(* Visualisation graf
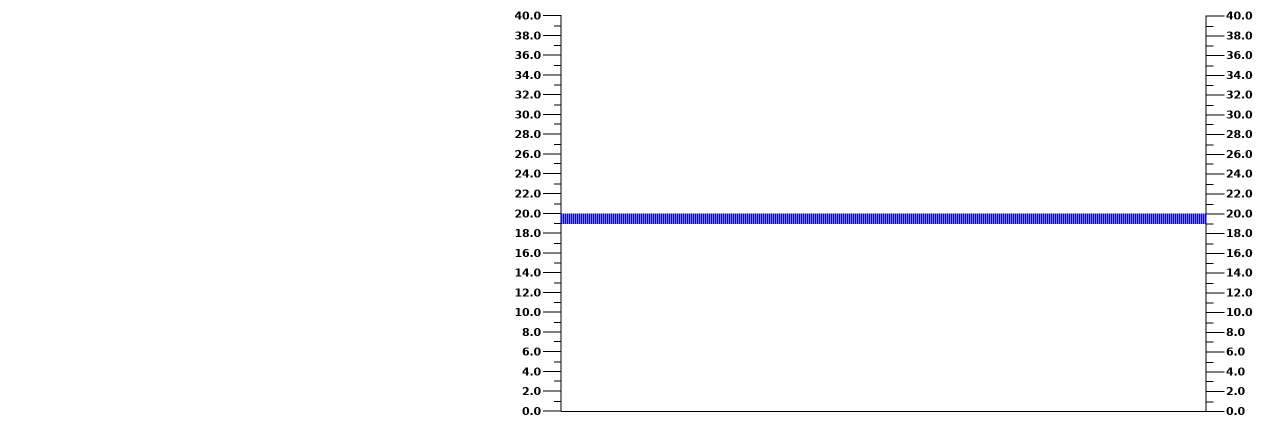
group at (130,90)-(861,501)
  rectangle at (0,8)-(1,9): text "{ExtendedElement},Visu\ElementDLL.ete,2,@Histogramm,731,411,PLC_PRG.test,,%.1f,1,2,0,40,0,0,0,0,0,0,0,-13,16,700,Arial,0,0,255,255,0,0,0,0,0,1,0.9,0_360,0,1,0,"
  rectangle at (0,411)-(25,427): text "0.0"
  rectangle at (706,411)-(731,427): text "0.0"
  rectangle at (0,390)-(25,406): text "2.0"
  rectangle at (706,390)-(731,406): text "2.0"
  rectangle at (0,370)-(25,386): text "4.0"
  rectangle at (706,370)-(731,386): text "4.0"
  rectangle at (0,349)-(25,365): text "6.0"
  rectangle at (706,349)-(731,365): text "6.0"
  rectangle at (0,329)-(25,345): text "8.0"
  rectangle at (706,329)-(731,345): text "8.0"
  rectangle at (0,308)-(25,324): text "10.0"
  rectangle at (706,308)-(731,324): text "10.0"
  rectangle at (0,288)-(25,304): text "12.0"
  rectangle at (706,288)-(731,304): text "12.0"
  rectangle at (0,267)-(25,283): text "14.0"
  rectangle at (706,267)-(731,283): text "14.0"
  rectangle at (0,247)-(25,263): text "16.0"
  rectangle at (706,247)-(731,263): text "16.0"
  rectangle at (0,226)-(25,242): text "18.0"
  rectangle at (706,226)-(731,242): text "18.0"
  rectangle at (0,206)-(25,222): text "20.0"
  rectangle at (706,206)-(731,222): text "20.0"
  rectangle at (0,185)-(25,201): text "22.0"
  rectangle at (706,185)-(731,201): text "22.0"
  rectangle at (0,164)-(25,180): text "24.0"
  rectangle at (706,164)-(731,180): text "24.0"
  rectangle at (0,144)-(25,160): text "26.0"
  rectangle at (706,144)-(731,160): text "26.0"
  rectangle at (0,123)-(25,139): text "28.0"
  rectangle at (706,123)-(731,139): text "28.0"
  rectangle at (0,103)-(25,119): text "30.0"
  rectangle at (706,103)-(731,119): text "30.0"
  rectangle at (0,82)-(25,98): text "32.0"
  rectangle at (706,82)-(731,98): text "32.0"
  rectangle at (0,62)-(25,78): text "34.0"
  rectangle at (706,62)-(731,78): text "34.0"
  rectangle at (0,41)-(25,57): text "36.0"
  rectangle at (706,41)-(731,57): text "36.0"
  rectangle at (0,21)-(25,37): text "38.0"
  rectangle at (706,21)-(731,37): text "38.0"
  rectangle at (0,0)-(25,16): text "40.0"
  rectangle at (706,0)-(731,16): text "40.0"
  rectangle at (43,214)-(44,224): alarm colour if PLC_PRG.test[0] < 0; top (-1.0 *  PLC_PRG.test[0]  +  20  ) * 10.275 + SEL( PLC_PRG.test[0] > 20 , 0.5, -0.5); bottom (-1.0 *  PLC_PRG.test[0]  +  20  ) * 10.275 + SEL( PLC_PRG.test[0] > 20 , 0.5, -0.5)
  rectangle at (45,214)-(46,224): alarm colour if PLC_PRG.test[1] < 0; top (-1.0 *  PLC_PRG.test[1]  +  20  ) * 10.275 + SEL( PLC_PRG.test[1] > 20 , 0.5, -0.5); bottom (-1.0 *  PLC_PRG.test[1]  +  20  ) * 10.275 + SEL( PLC_PRG.test[1] > 20 , 0.5, -0.5)
  rectangle at (47,214)-(48,224): alarm colour if PLC_PRG.test[2] < 0; top (-1.0 *  PLC_PRG.test[2]  +  20  ) * 10.275 + SEL( PLC_PRG.test[2] > 20 , 0.5, -0.5); bottom (-1.0 *  PLC_PRG.test[2]  +  20  ) * 10.275 + SEL( PLC_PRG.test[2] > 20 , 0.5, -0.5)
  rectangle at (49,214)-(50,224): alarm colour if PLC_PRG.test[3] < 0; top (-1.0 *  PLC_PRG.test[3]  +  20  ) * 10.275 + SEL( PLC_PRG.test[3] > 20 , 0.5, -0.5); bottom (-1.0 *  PLC_PRG.test[3]  +  20  ) * 10.275 + SEL( PLC_PRG.test[3] > 20 , 0.5, -0.5)
  rectangle at (51,214)-(52,224): alarm colour if PLC_PRG.test[4] < 0; top (-1.0 *  PLC_PRG.test[4]  +  20  ) * 10.275 + SEL( PLC_PRG.test[4] > 20 , 0.5, -0.5); bottom (-1.0 *  PLC_PRG.test[4]  +  20  ) * 10.275 + SEL( PLC_PRG.test[4] > 20 , 0.5, -0.5)
  rectangle at (53,214)-(54,224): alarm colour if PLC_PRG.test[5] < 0; top (-1.0 *  PLC_PRG.test[5]  +  20  ) * 10.275 + SEL( PLC_PRG.test[5] > 20 , 0.5, -0.5); bottom (-1.0 *  PLC_PRG.test[5]  +  20  ) * 10.275 + SEL( PLC_PRG.test[5] > 20 , 0.5, -0.5)
  rectangle at (55,214)-(56,224): alarm colour if PLC_PRG.test[6] < 0; top (-1.0 *  PLC_PRG.test[6]  +  20  ) * 10.275 + SEL( PLC_PRG.test[6] > 20 , 0.5, -0.5); bottom (-1.0 *  PLC_PRG.test[6]  +  20  ) * 10.275 + SEL( PLC_PRG.test[6] > 20 , 0.5, -0.5)
  rectangle at (57,214)-(58,224): alarm colour if PLC_PRG.test[7] < 0; top (-1.0 *  PLC_PRG.test[7]  +  20  ) * 10.275 + SEL( PLC_PRG.test[7] > 20 , 0.5, -0.5); bottom (-1.0 *  PLC_PRG.test[7]  +  20  ) * 10.275 + SEL( PLC_PRG.test[7] > 20 , 0.5, -0.5)
  rectangle at (59,214)-(60,224): alarm colour if PLC_PRG.test[8] < 0; top (-1.0 *  PLC_PRG.test[8]  +  20  ) * 10.275 + SEL( PLC_PRG.test[8] > 20 , 0.5, -0.5); bottom (-1.0 *  PLC_PRG.test[8]  +  20  ) * 10.275 + SEL( PLC_PRG.test[8] > 20 , 0.5, -0.5)
  rectangle at (61,214)-(62,224): alarm colour if PLC_PRG.test[9] < 0; top (-1.0 *  PLC_PRG.test[9]  +  20  ) * 10.275 + SEL( PLC_PRG.test[9] > 20 , 0.5, -0.5); bottom (-1.0 *  PLC_PRG.test[9]  +  20  ) * 10.275 + SEL( PLC_PRG.test[9] > 20 , 0.5, -0.5)
  rectangle at (63,214)-(64,224): alarm colour if PLC_PRG.test[10] < 0; top (-1.0 *  PLC_PRG.test[10]  +  20  ) * 10.275 + SEL( PLC_PRG.test[10] > 20 , 0.5, -0.5); bottom (-1.0 *  PLC_PRG.test[10]  +  20  ) * 10.275 + SEL( PLC_PRG.test[10] > 20 , 0.5, -0.5)
  rectangle at (65,214)-(66,224): alarm colour if PLC_PRG.test[11] < 0; top (-1.0 *  PLC_PRG.test[11]  +  20  ) * 10.275 + SEL( PLC_PRG.test[11] > 20 , 0.5, -0.5); bottom (-1.0 *  PLC_PRG.test[11]  +  20  ) * 10.275 + SEL( PLC_PRG.test[11] > 20 , 0.5, -0.5)
  rectangle at (67,214)-(68,224): alarm colour if PLC_PRG.test[12] < 0; top (-1.0 *  PLC_PRG.test[12]  +  20  ) * 10.275 + SEL( PLC_PRG.test[12] > 20 , 0.5, -0.5); bottom (-1.0 *  PLC_PRG.test[12]  +  20  ) * 10.275 + SEL( PLC_PRG.test[12] > 20 , 0.5, -0.5)
  rectangle at (69,214)-(70,224): alarm colour if PLC_PRG.test[13] < 0; top (-1.0 *  PLC_PRG.test[13]  +  20  ) * 10.275 + SEL( PLC_PRG.test[13] > 20 , 0.5, -0.5); bottom (-1.0 *  PLC_PRG.test[13]  +  20  ) * 10.275 + SEL( PLC_PRG.test[13] > 20 , 0.5, -0.5)
  rectangle at (71,214)-(72,224): alarm colour if PLC_PRG.test[14] < 0; top (-1.0 *  PLC_PRG.test[14]  +  20  ) * 10.275 + SEL( PLC_PRG.test[14] > 20 , 0.5, -0.5); bottom (-1.0 *  PLC_PRG.test[14]  +  20  ) * 10.275 + SEL( PLC_PRG.test[14] > 20 , 0.5, -0.5)
  rectangle at (73,214)-(74,224): alarm colour if PLC_PRG.test[15] < 0; top (-1.0 *  PLC_PRG.test[15]  +  20  ) * 10.275 + SEL( PLC_PRG.test[15] > 20 , 0.5, -0.5); bottom (-1.0 *  PLC_PRG.test[15]  +  20  ) * 10.275 + SEL( PLC_PRG.test[15] > 20 , 0.5, -0.5)
  rectangle at (75,214)-(76,224): alarm colour if PLC_PRG.test[16] < 0; top (-1.0 *  PLC_PRG.test[16]  +  20  ) * 10.275 + SEL( PLC_PRG.test[16] > 20 , 0.5, -0.5); bottom (-1.0 *  PLC_PRG.test[16]  +  20  ) * 10.275 + SEL( PLC_PRG.test[16] > 20 , 0.5, -0.5)
  rectangle at (77,214)-(78,224): alarm colour if PLC_PRG.test[17] < 0; top (-1.0 *  PLC_PRG.test[17]  +  20  ) * 10.275 + SEL( PLC_PRG.test[17] > 20 , 0.5, -0.5); bottom (-1.0 *  PLC_PRG.test[17]  +  20  ) * 10.275 + SEL( PLC_PRG.test[17] > 20 , 0.5, -0.5)
  rectangle at (79,214)-(80,224): alarm colour if PLC_PRG.test[18] < 0; top (-1.0 *  PLC_PRG.test[18]  +  20  ) * 10.275 + SEL( PLC_PRG.test[18] > 20 , 0.5, -0.5); bottom (-1.0 *  PLC_PRG.test[18]  +  20  ) * 10.275 + SEL( PLC_PRG.test[18] > 20 , 0.5, -0.5)
  rectangle at (81,214)-(82,224): alarm colour if PLC_PRG.test[19] < 0; top (-1.0 *  PLC_PRG.test[19]  +  20  ) * 10.275 + SEL( PLC_PRG.test[19] > 20 , 0.5, -0.5); bottom (-1.0 *  PLC_PRG.test[19]  +  20  ) * 10.275 + SEL( PLC_PRG.test[19] > 20 , 0.5, -0.5)
  rectangle at (83,214)-(84,224): alarm colour if PLC_PRG.test[20] < 0; top (-1.0 *  PLC_PRG.test[20]  +  20  ) * 10.275 + SEL( PLC_PRG.test[20] > 20 , 0.5, -0.5); bottom (-1.0 *  PLC_PRG.test[20]  +  20  ) * 10.275 + SEL( PLC_PRG.test[20] > 20 , 0.5, -0.5)
  rectangle at (85,214)-(86,224): alarm colour if PLC_PRG.test[21] < 0; top (-1.0 *  PLC_PRG.test[21]  +  20  ) * 10.275 + SEL( PLC_PRG.test[21] > 20 , 0.5, -0.5); bottom (-1.0 *  PLC_PRG.test[21]  +  20  ) * 10.275 + SEL( PLC_PRG.test[21] > 20 , 0.5, -0.5)
  rectangle at (87,214)-(88,224): alarm colour if PLC_PRG.test[22] < 0; top (-1.0 *  PLC_PRG.test[22]  +  20  ) * 10.275 + SEL( PLC_PRG.test[22] > 20 , 0.5, -0.5); bottom (-1.0 *  PLC_PRG.test[22]  +  20  ) * 10.275 + SEL( PLC_PRG.test[22] > 20 , 0.5, -0.5)
  rectangle at (89,214)-(90,224): alarm colour if PLC_PRG.test[23] < 0; top (-1.0 *  PLC_PRG.test[23]  +  20  ) * 10.275 + SEL( PLC_PRG.test[23] > 20 , 0.5, -0.5); bottom (-1.0 *  PLC_PRG.test[23]  +  20  ) * 10.275 + SEL( PLC_PRG.test[23] > 20 , 0.5, -0.5)
  rectangle at (91,214)-(92,224): alarm colour if PLC_PRG.test[24] < 0; top (-1.0 *  PLC_PRG.test[24]  +  20  ) * 10.275 + SEL( PLC_PRG.test[24] > 20 , 0.5, -0.5); bottom (-1.0 *  PLC_PRG.test[24]  +  20  ) * 10.275 + SEL( PLC_PRG.test[24] > 20 , 0.5, -0.5)
  rectangle at (93,214)-(94,224): alarm colour if PLC_PRG.test[25] < 0; top (-1.0 *  PLC_PRG.test[25]  +  20  ) * 10.275 + SEL( PLC_PRG.test[25] > 20 , 0.5, -0.5); bottom (-1.0 *  PLC_PRG.test[25]  +  20  ) * 10.275 + SEL( PLC_PRG.test[25] > 20 , 0.5, -0.5)
  rectangle at (95,214)-(96,224): alarm colour if PLC_PRG.test[26] < 0; top (-1.0 *  PLC_PRG.test[26]  +  20  ) * 10.275 + SEL( PLC_PRG.test[26] > 20 , 0.5, -0.5); bottom (-1.0 *  PLC_PRG.test[26]  +  20  ) * 10.275 + SEL( PLC_PRG.test[26] > 20 , 0.5, -0.5)
  rectangle at (97,214)-(98,224): alarm colour if PLC_PRG.test[27] < 0; top (-1.0 *  PLC_PRG.test[27]  +  20  ) * 10.275 + SEL( PLC_PRG.test[27] > 20 , 0.5, -0.5); bottom (-1.0 *  PLC_PRG.test[27]  +  20  ) * 10.275 + SEL( PLC_PRG.test[27] > 20 , 0.5, -0.5)
  rectangle at (99,214)-(100,224): alarm colour if PLC_PRG.test[28] < 0; top (-1.0 *  PLC_PRG.test[28]  +  20  ) * 10.275 + SEL( PLC_PRG.test[28] > 20 , 0.5, -0.5); bottom (-1.0 *  PLC_PRG.test[28]  +  20  ) * 10.275 + SEL( PLC_PRG.test[28] > 20 , 0.5, -0.5)
  rectangle at (101,214)-(102,224): alarm colour if PLC_PRG.test[29] < 0; top (-1.0 *  PLC_PRG.test[29]  +  20  ) * 10.275 + SEL( PLC_PRG.test[29] > 20 , 0.5, -0.5); bottom (-1.0 *  PLC_PRG.test[29]  +  20  ) * 10.275 + SEL( PLC_PRG.test[29] > 20 , 0.5, -0.5)
  rectangle at (103,214)-(104,224): alarm colour if PLC_PRG.test[30] < 0; top (-1.0 *  PLC_PRG.test[30]  +  20  ) * 10.275 + SEL( PLC_PRG.test[30] > 20 , 0.5, -0.5); bottom (-1.0 *  PLC_PRG.test[30]  +  20  ) * 10.275 + SEL( PLC_PRG.test[30] > 20 , 0.5, -0.5)
  rectangle at (105,214)-(106,224): alarm colour if PLC_PRG.test[31] < 0; top (-1.0 *  PLC_PRG.test[31]  +  20  ) * 10.275 + SEL( PLC_PRG.test[31] > 20 , 0.5, -0.5); bottom (-1.0 *  PLC_PRG.test[31]  +  20  ) * 10.275 + SEL( PLC_PRG.test[31] > 20 , 0.5, -0.5)
  rectangle at (107,214)-(108,224): alarm colour if PLC_PRG.test[32] < 0; top (-1.0 *  PLC_PRG.test[32]  +  20  ) * 10.275 + SEL( PLC_PRG.test[32] > 20 , 0.5, -0.5); bottom (-1.0 *  PLC_PRG.test[32]  +  20  ) * 10.275 + SEL( PLC_PRG.test[32] > 20 , 0.5, -0.5)
  rectangle at (109,214)-(110,224): alarm colour if PLC_PRG.test[33] < 0; top (-1.0 *  PLC_PRG.test[33]  +  20  ) * 10.275 + SEL( PLC_PRG.test[33] > 20 , 0.5, -0.5); bottom (-1.0 *  PLC_PRG.test[33]  +  20  ) * 10.275 + SEL( PLC_PRG.test[33] > 20 , 0.5, -0.5)
  rectangle at (111,214)-(112,224): alarm colour if PLC_PRG.test[34] < 0; top (-1.0 *  PLC_PRG.test[34]  +  20  ) * 10.275 + SEL( PLC_PRG.test[34] > 20 , 0.5, -0.5); bottom (-1.0 *  PLC_PRG.test[34]  +  20  ) * 10.275 + SEL( PLC_PRG.test[34] > 20 , 0.5, -0.5)
  rectangle at (113,214)-(114,224): alarm colour if PLC_PRG.test[35] < 0; top (-1.0 *  PLC_PRG.test[35]  +  20  ) * 10.275 + SEL( PLC_PRG.test[35] > 20 , 0.5, -0.5); bottom (-1.0 *  PLC_PRG.test[35]  +  20  ) * 10.275 + SEL( PLC_PRG.test[35] > 20 , 0.5, -0.5)
  rectangle at (115,214)-(116,224): alarm colour if PLC_PRG.test[36] < 0; top (-1.0 *  PLC_PRG.test[36]  +  20  ) * 10.275 + SEL( PLC_PRG.test[36] > 20 , 0.5, -0.5); bottom (-1.0 *  PLC_PRG.test[36]  +  20  ) * 10.275 + SEL( PLC_PRG.test[36] > 20 , 0.5, -0.5)
  rectangle at (117,214)-(118,224): alarm colour if PLC_PRG.test[37] < 0; top (-1.0 *  PLC_PRG.test[37]  +  20  ) * 10.275 + SEL( PLC_PRG.test[37] > 20 , 0.5, -0.5); bottom (-1.0 *  PLC_PRG.test[37]  +  20  ) * 10.275 + SEL( PLC_PRG.test[37] > 20 , 0.5, -0.5)
  rectangle at (119,214)-(120,224): alarm colour if PLC_PRG.test[38] < 0; top (-1.0 *  PLC_PRG.test[38]  +  20  ) * 10.275 + SEL( PLC_PRG.test[38] > 20 , 0.5, -0.5); bottom (-1.0 *  PLC_PRG.test[38]  +  20  ) * 10.275 + SEL( PLC_PRG.test[38] > 20 , 0.5, -0.5)
  rectangle at (121,214)-(122,224): alarm colour if PLC_PRG.test[39] < 0; top (-1.0 *  PLC_PRG.test[39]  +  20  ) * 10.275 + SEL( PLC_PRG.test[39] > 20 , 0.5, -0.5); bottom (-1.0 *  PLC_PRG.test[39]  +  20  ) * 10.275 + SEL( PLC_PRG.test[39] > 20 , 0.5, -0.5)
  rectangle at (123,214)-(124,224): alarm colour if PLC_PRG.test[40] < 0; top (-1.0 *  PLC_PRG.test[40]  +  20  ) * 10.275 + SEL( PLC_PRG.test[40] > 20 , 0.5, -0.5); bottom (-1.0 *  PLC_PRG.test[40]  +  20  ) * 10.275 + SEL( PLC_PRG.test[40] > 20 , 0.5, -0.5)
  rectangle at (125,214)-(126,224): alarm colour if PLC_PRG.test[41] < 0; top (-1.0 *  PLC_PRG.test[41]  +  20  ) * 10.275 + SEL( PLC_PRG.test[41] > 20 , 0.5, -0.5); bottom (-1.0 *  PLC_PRG.test[41]  +  20  ) * 10.275 + SEL( PLC_PRG.test[41] > 20 , 0.5, -0.5)
  rectangle at (127,214)-(128,224): alarm colour if PLC_PRG.test[42] < 0; top (-1.0 *  PLC_PRG.test[42]  +  20  ) * 10.275 + SEL( PLC_PRG.test[42] > 20 , 0.5, -0.5); bottom (-1.0 *  PLC_PRG.test[42]  +  20  ) * 10.275 + SEL( PLC_PRG.test[42] > 20 , 0.5, -0.5)
  rectangle at (129,214)-(130,224): alarm colour if PLC_PRG.test[43] < 0; top (-1.0 *  PLC_PRG.test[43]  +  20  ) * 10.275 + SEL( PLC_PRG.test[43] > 20 , 0.5, -0.5); bottom (-1.0 *  PLC_PRG.test[43]  +  20  ) * 10.275 + SEL( PLC_PRG.test[43] > 20 , 0.5, -0.5)
  rectangle at (131,214)-(132,224): alarm colour if PLC_PRG.test[44] < 0; top (-1.0 *  PLC_PRG.test[44]  +  20  ) * 10.275 + SEL( PLC_PRG.test[44] > 20 , 0.5, -0.5); bottom (-1.0 *  PLC_PRG.test[44]  +  20  ) * 10.275 + SEL( PLC_PRG.test[44] > 20 , 0.5, -0.5)
  rectangle at (133,214)-(134,224): alarm colour if PLC_PRG.test[45] < 0; top (-1.0 *  PLC_PRG.test[45]  +  20  ) * 10.275 + SEL( PLC_PRG.test[45] > 20 , 0.5, -0.5); bottom (-1.0 *  PLC_PRG.test[45]  +  20  ) * 10.275 + SEL( PLC_PRG.test[45] > 20 , 0.5, -0.5)
  rectangle at (135,214)-(136,224): alarm colour if PLC_PRG.test[46] < 0; top (-1.0 *  PLC_PRG.test[46]  +  20  ) * 10.275 + SEL( PLC_PRG.test[46] > 20 , 0.5, -0.5); bottom (-1.0 *  PLC_PRG.test[46]  +  20  ) * 10.275 + SEL( PLC_PRG.test[46] > 20 , 0.5, -0.5)
  rectangle at (137,214)-(138,224): alarm colour if PLC_PRG.test[47] < 0; top (-1.0 *  PLC_PRG.test[47]  +  20  ) * 10.275 + SEL( PLC_PRG.test[47] > 20 , 0.5, -0.5); bottom (-1.0 *  PLC_PRG.test[47]  +  20  ) * 10.275 + SEL( PLC_PRG.test[47] > 20 , 0.5, -0.5)
  rectangle at (139,214)-(140,224): alarm colour if PLC_PRG.test[48] < 0; top (-1.0 *  PLC_PRG.test[48]  +  20  ) * 10.275 + SEL( PLC_PRG.test[48] > 20 , 0.5, -0.5); bottom (-1.0 *  PLC_PRG.test[48]  +  20  ) * 10.275 + SEL( PLC_PRG.test[48] > 20 , 0.5, -0.5)
  rectangle at (141,214)-(142,224): alarm colour if PLC_PRG.test[49] < 0; top (-1.0 *  PLC_PRG.test[49]  +  20  ) * 10.275 + SEL( PLC_PRG.test[49] > 20 , 0.5, -0.5); bottom (-1.0 *  PLC_PRG.test[49]  +  20  ) * 10.275 + SEL( PLC_PRG.test[49] > 20 , 0.5, -0.5)
  rectangle at (143,214)-(144,224): alarm colour if PLC_PRG.test[50] < 0; top (-1.0 *  PLC_PRG.test[50]  +  20  ) * 10.275 + SEL( PLC_PRG.test[50] > 20 , 0.5, -0.5); bottom (-1.0 *  PLC_PRG.test[50]  +  20  ) * 10.275 + SEL( PLC_PRG.test[50] > 20 , 0.5, -0.5)
  rectangle at (145,214)-(146,224): alarm colour if PLC_PRG.test[51] < 0; top (-1.0 *  PLC_PRG.test[51]  +  20  ) * 10.275 + SEL( PLC_PRG.test[51] > 20 , 0.5, -0.5); bottom (-1.0 *  PLC_PRG.test[51]  +  20  ) * 10.275 + SEL( PLC_PRG.test[51] > 20 , 0.5, -0.5)
  rectangle at (147,214)-(148,224): alarm colour if PLC_PRG.test[52] < 0; top (-1.0 *  PLC_PRG.test[52]  +  20  ) * 10.275 + SEL( PLC_PRG.test[52] > 20 , 0.5, -0.5); bottom (-1.0 *  PLC_PRG.test[52]  +  20  ) * 10.275 + SEL( PLC_PRG.test[52] > 20 , 0.5, -0.5)
  rectangle at (149,214)-(150,224): alarm colour if PLC_PRG.test[53] < 0; top (-1.0 *  PLC_PRG.test[53]  +  20  ) * 10.275 + SEL( PLC_PRG.test[53] > 20 , 0.5, -0.5); bottom (-1.0 *  PLC_PRG.test[53]  +  20  ) * 10.275 + SEL( PLC_PRG.test[53] > 20 , 0.5, -0.5)
  rectangle at (151,214)-(152,224): alarm colour if PLC_PRG.test[54] < 0; top (-1.0 *  PLC_PRG.test[54]  +  20  ) * 10.275 + SEL( PLC_PRG.test[54] > 20 , 0.5, -0.5); bottom (-1.0 *  PLC_PRG.test[54]  +  20  ) * 10.275 + SEL( PLC_PRG.test[54] > 20 , 0.5, -0.5)
  rectangle at (153,214)-(154,224): alarm colour if PLC_PRG.test[55] < 0; top (-1.0 *  PLC_PRG.test[55]  +  20  ) * 10.275 + SEL( PLC_PRG.test[55] > 20 , 0.5, -0.5); bottom (-1.0 *  PLC_PRG.test[55]  +  20  ) * 10.275 + SEL( PLC_PRG.test[55] > 20 , 0.5, -0.5)
  rectangle at (155,214)-(156,224): alarm colour if PLC_PRG.test[56] < 0; top (-1.0 *  PLC_PRG.test[56]  +  20  ) * 10.275 + SEL( PLC_PRG.test[56] > 20 , 0.5, -0.5); bottom (-1.0 *  PLC_PRG.test[56]  +  20  ) * 10.275 + SEL( PLC_PRG.test[56] > 20 , 0.5, -0.5)
  rectangle at (157,214)-(158,224): alarm colour if PLC_PRG.test[57] < 0; top (-1.0 *  PLC_PRG.test[57]  +  20  ) * 10.275 + SEL( PLC_PRG.test[57] > 20 , 0.5, -0.5); bottom (-1.0 *  PLC_PRG.test[57]  +  20  ) * 10.275 + SEL( PLC_PRG.test[57] > 20 , 0.5, -0.5)
  rectangle at (159,214)-(160,224): alarm colour if PLC_PRG.test[58] < 0; top (-1.0 *  PLC_PRG.test[58]  +  20  ) * 10.275 + SEL( PLC_PRG.test[58] > 20 , 0.5, -0.5); bottom (-1.0 *  PLC_PRG.test[58]  +  20  ) * 10.275 + SEL( PLC_PRG.test[58] > 20 , 0.5, -0.5)
  rectangle at (161,214)-(162,224): alarm colour if PLC_PRG.test[59] < 0; top (-1.0 *  PLC_PRG.test[59]  +  20  ) * 10.275 + SEL( PLC_PRG.test[59] > 20 , 0.5, -0.5); bottom (-1.0 *  PLC_PRG.test[59]  +  20  ) * 10.275 + SEL( PLC_PRG.test[59] > 20 , 0.5, -0.5)
  rectangle at (163,214)-(164,224): alarm colour if PLC_PRG.test[60] < 0; top (-1.0 *  PLC_PRG.test[60]  +  20  ) * 10.275 + SEL( PLC_PRG.test[60] > 20 , 0.5, -0.5); bottom (-1.0 *  PLC_PRG.test[60]  +  20  ) * 10.275 + SEL( PLC_PRG.test[60] > 20 , 0.5, -0.5)
  rectangle at (165,214)-(166,224): alarm colour if PLC_PRG.test[61] < 0; top (-1.0 *  PLC_PRG.test[61]  +  20  ) * 10.275 + SEL( PLC_PRG.test[61] > 20 , 0.5, -0.5); bottom (-1.0 *  PLC_PRG.test[61]  +  20  ) * 10.275 + SEL( PLC_PRG.test[61] > 20 , 0.5, -0.5)
  rectangle at (167,214)-(168,224): alarm colour if PLC_PRG.test[62] < 0; top (-1.0 *  PLC_PRG.test[62]  +  20  ) * 10.275 + SEL( PLC_PRG.test[62] > 20 , 0.5, -0.5); bottom (-1.0 *  PLC_PRG.test[62]  +  20  ) * 10.275 + SEL( PLC_PRG.test[62] > 20 , 0.5, -0.5)
  rectangle at (169,214)-(170,224): alarm colour if PLC_PRG.test[63] < 0; top (-1.0 *  PLC_PRG.test[63]  +  20  ) * 10.275 + SEL( PLC_PRG.test[63] > 20 , 0.5, -0.5); bottom (-1.0 *  PLC_PRG.test[63]  +  20  ) * 10.275 + SEL( PLC_PRG.test[63] > 20 , 0.5, -0.5)
  rectangle at (171,214)-(172,224): alarm colour if PLC_PRG.test[64] < 0; top (-1.0 *  PLC_PRG.test[64]  +  20  ) * 10.275 + SEL( PLC_PRG.test[64] > 20 , 0.5, -0.5); bottom (-1.0 *  PLC_PRG.test[64]  +  20  ) * 10.275 + SEL( PLC_PRG.test[64] > 20 , 0.5, -0.5)
  rectangle at (173,214)-(174,224): alarm colour if PLC_PRG.test[65] < 0; top (-1.0 *  PLC_PRG.test[65]  +  20  ) * 10.275 + SEL( PLC_PRG.test[65] > 20 , 0.5, -0.5); bottom (-1.0 *  PLC_PRG.test[65]  +  20  ) * 10.275 + SEL( PLC_PRG.test[65] > 20 , 0.5, -0.5)
  rectangle at (175,214)-(176,224): alarm colour if PLC_PRG.test[66] < 0; top (-1.0 *  PLC_PRG.test[66]  +  20  ) * 10.275 + SEL( PLC_PRG.test[66] > 20 , 0.5, -0.5); bottom (-1.0 *  PLC_PRG.test[66]  +  20  ) * 10.275 + SEL( PLC_PRG.test[66] > 20 , 0.5, -0.5)
  rectangle at (177,214)-(178,224): alarm colour if PLC_PRG.test[67] < 0; top (-1.0 *  PLC_PRG.test[67]  +  20  ) * 10.275 + SEL( PLC_PRG.test[67] > 20 , 0.5, -0.5); bottom (-1.0 *  PLC_PRG.test[67]  +  20  ) * 10.275 + SEL( PLC_PRG.test[67] > 20 , 0.5, -0.5)
  rectangle at (179,214)-(180,224): alarm colour if PLC_PRG.test[68] < 0; top (-1.0 *  PLC_PRG.test[68]  +  20  ) * 10.275 + SEL( PLC_PRG.test[68] > 20 , 0.5, -0.5); bottom (-1.0 *  PLC_PRG.test[68]  +  20  ) * 10.275 + SEL( PLC_PRG.test[68] > 20 , 0.5, -0.5)
  rectangle at (181,214)-(182,224): alarm colour if PLC_PRG.test[69] < 0; top (-1.0 *  PLC_PRG.test[69]  +  20  ) * 10.275 + SEL( PLC_PRG.test[69] > 20 , 0.5, -0.5); bottom (-1.0 *  PLC_PRG.test[69]  +  20  ) * 10.275 + SEL( PLC_PRG.test[69] > 20 , 0.5, -0.5)
  rectangle at (183,214)-(184,224): alarm colour if PLC_PRG.test[70] < 0; top (-1.0 *  PLC_PRG.test[70]  +  20  ) * 10.275 + SEL( PLC_PRG.test[70] > 20 , 0.5, -0.5); bottom (-1.0 *  PLC_PRG.test[70]  +  20  ) * 10.275 + SEL( PLC_PRG.test[70] > 20 , 0.5, -0.5)
  rectangle at (185,214)-(186,224): alarm colour if PLC_PRG.test[71] < 0; top (-1.0 *  PLC_PRG.test[71]  +  20  ) * 10.275 + SEL( PLC_PRG.test[71] > 20 , 0.5, -0.5); bottom (-1.0 *  PLC_PRG.test[71]  +  20  ) * 10.275 + SEL( PLC_PRG.test[71] > 20 , 0.5, -0.5)
  rectangle at (187,214)-(188,224): alarm colour if PLC_PRG.test[72] < 0; top (-1.0 *  PLC_PRG.test[72]  +  20  ) * 10.275 + SEL( PLC_PRG.test[72] > 20 , 0.5, -0.5); bottom (-1.0 *  PLC_PRG.test[72]  +  20  ) * 10.275 + SEL( PLC_PRG.test[72] > 20 , 0.5, -0.5)
  rectangle at (189,214)-(190,224): alarm colour if PLC_PRG.test[73] < 0; top (-1.0 *  PLC_PRG.test[73]  +  20  ) * 10.275 + SEL( PLC_PRG.test[73] > 20 , 0.5, -0.5); bottom (-1.0 *  PLC_PRG.test[73]  +  20  ) * 10.275 + SEL( PLC_PRG.test[73] > 20 , 0.5, -0.5)
  rectangle at (191,214)-(192,224): alarm colour if PLC_PRG.test[74] < 0; top (-1.0 *  PLC_PRG.test[74]  +  20  ) * 10.275 + SEL( PLC_PRG.test[74] > 20 , 0.5, -0.5); bottom (-1.0 *  PLC_PRG.test[74]  +  20  ) * 10.275 + SEL( PLC_PRG.test[74] > 20 , 0.5, -0.5)
  rectangle at (193,214)-(194,224): alarm colour if PLC_PRG.test[75] < 0; top (-1.0 *  PLC_PRG.test[75]  +  20  ) * 10.275 + SEL( PLC_PRG.test[75] > 20 , 0.5, -0.5); bottom (-1.0 *  PLC_PRG.test[75]  +  20  ) * 10.275 + SEL( PLC_PRG.test[75] > 20 , 0.5, -0.5)
  rectangle at (195,214)-(196,224): alarm colour if PLC_PRG.test[76] < 0; top (-1.0 *  PLC_PRG.test[76]  +  20  ) * 10.275 + SEL( PLC_PRG.test[76] > 20 , 0.5, -0.5); bottom (-1.0 *  PLC_PRG.test[76]  +  20  ) * 10.275 + SEL( PLC_PRG.test[76] > 20 , 0.5, -0.5)
  rectangle at (197,214)-(198,224): alarm colour if PLC_PRG.test[77] < 0; top (-1.0 *  PLC_PRG.test[77]  +  20  ) * 10.275 + SEL( PLC_PRG.test[77] > 20 , 0.5, -0.5); bottom (-1.0 *  PLC_PRG.test[77]  +  20  ) * 10.275 + SEL( PLC_PRG.test[77] > 20 , 0.5, -0.5)
  rectangle at (199,214)-(200,224): alarm colour if PLC_PRG.test[78] < 0; top (-1.0 *  PLC_PRG.test[78]  +  20  ) * 10.275 + SEL( PLC_PRG.test[78] > 20 , 0.5, -0.5); bottom (-1.0 *  PLC_PRG.test[78]  +  20  ) * 10.275 + SEL( PLC_PRG.test[78] > 20 , 0.5, -0.5)
  rectangle at (201,214)-(202,224): alarm colour if PLC_PRG.test[79] < 0; top (-1.0 *  PLC_PRG.test[79]  +  20  ) * 10.275 + SEL( PLC_PRG.test[79] > 20 , 0.5, -0.5); bottom (-1.0 *  PLC_PRG.test[79]  +  20  ) * 10.275 + SEL( PLC_PRG.test[79] > 20 , 0.5, -0.5)
  rectangle at (203,214)-(204,224): alarm colour if PLC_PRG.test[80] < 0; top (-1.0 *  PLC_PRG.test[80]  +  20  ) * 10.275 + SEL( PLC_PRG.test[80] > 20 , 0.5, -0.5); bottom (-1.0 *  PLC_PRG.test[80]  +  20  ) * 10.275 + SEL( PLC_PRG.test[80] > 20 , 0.5, -0.5)
  rectangle at (205,214)-(206,224): alarm colour if PLC_PRG.test[81] < 0; top (-1.0 *  PLC_PRG.test[81]  +  20  ) * 10.275 + SEL( PLC_PRG.test[81] > 20 , 0.5, -0.5); bottom (-1.0 *  PLC_PRG.test[81]  +  20  ) * 10.275 + SEL( PLC_PRG.test[81] > 20 , 0.5, -0.5)
  rectangle at (207,214)-(208,224): alarm colour if PLC_PRG.test[82] < 0; top (-1.0 *  PLC_PRG.test[82]  +  20  ) * 10.275 + SEL( PLC_PRG.test[82] > 20 , 0.5, -0.5); bottom (-1.0 *  PLC_PRG.test[82]  +  20  ) * 10.275 + SEL( PLC_PRG.test[82] > 20 , 0.5, -0.5)
  rectangle at (209,214)-(210,224): alarm colour if PLC_PRG.test[83] < 0; top (-1.0 *  PLC_PRG.test[83]  +  20  ) * 10.275 + SEL( PLC_PRG.test[83] > 20 , 0.5, -0.5); bottom (-1.0 *  PLC_PRG.test[83]  +  20  ) * 10.275 + SEL( PLC_PRG.test[83] > 20 , 0.5, -0.5)
  rectangle at (211,214)-(212,224): alarm colour if PLC_PRG.test[84] < 0; top (-1.0 *  PLC_PRG.test[84]  +  20  ) * 10.275 + SEL( PLC_PRG.test[84] > 20 , 0.5, -0.5); bottom (-1.0 *  PLC_PRG.test[84]  +  20  ) * 10.275 + SEL( PLC_PRG.test[84] > 20 , 0.5, -0.5)
  rectangle at (213,214)-(214,224): alarm colour if PLC_PRG.test[85] < 0; top (-1.0 *  PLC_PRG.test[85]  +  20  ) * 10.275 + SEL( PLC_PRG.test[85] > 20 , 0.5, -0.5); bottom (-1.0 *  PLC_PRG.test[85]  +  20  ) * 10.275 + SEL( PLC_PRG.test[85] > 20 , 0.5, -0.5)
  rectangle at (215,214)-(216,224): alarm colour if PLC_PRG.test[86] < 0; top (-1.0 *  PLC_PRG.test[86]  +  20  ) * 10.275 + SEL( PLC_PRG.test[86] > 20 , 0.5, -0.5); bottom (-1.0 *  PLC_PRG.test[86]  +  20  ) * 10.275 + SEL( PLC_PRG.test[86] > 20 , 0.5, -0.5)
  rectangle at (217,214)-(218,224): alarm colour if PLC_PRG.test[87] < 0; top (-1.0 *  PLC_PRG.test[87]  +  20  ) * 10.275 + SEL( PLC_PRG.test[87] > 20 , 0.5, -0.5); bottom (-1.0 *  PLC_PRG.test[87]  +  20  ) * 10.275 + SEL( PLC_PRG.test[87] > 20 , 0.5, -0.5)
  rectangle at (219,214)-(220,224): alarm colour if PLC_PRG.test[88] < 0; top (-1.0 *  PLC_PRG.test[88]  +  20  ) * 10.275 + SEL( PLC_PRG.test[88] > 20 , 0.5, -0.5); bottom (-1.0 *  PLC_PRG.test[88]  +  20  ) * 10.275 + SEL( PLC_PRG.test[88] > 20 , 0.5, -0.5)
  rectangle at (221,214)-(222,224): alarm colour if PLC_PRG.test[89] < 0; top (-1.0 *  PLC_PRG.test[89]  +  20  ) * 10.275 + SEL( PLC_PRG.test[89] > 20 , 0.5, -0.5); bottom (-1.0 *  PLC_PRG.test[89]  +  20  ) * 10.275 + SEL( PLC_PRG.test[89] > 20 , 0.5, -0.5)
  rectangle at (223,214)-(224,224): alarm colour if PLC_PRG.test[90] < 0; top (-1.0 *  PLC_PRG.test[90]  +  20  ) * 10.275 + SEL( PLC_PRG.test[90] > 20 , 0.5, -0.5); bottom (-1.0 *  PLC_PRG.test[90]  +  20  ) * 10.275 + SEL( PLC_PRG.test[90] > 20 , 0.5, -0.5)
  rectangle at (225,214)-(226,224): alarm colour if PLC_PRG.test[91] < 0; top (-1.0 *  PLC_PRG.test[91]  +  20  ) * 10.275 + SEL( PLC_PRG.test[91] > 20 , 0.5, -0.5); bottom (-1.0 *  PLC_PRG.test[91]  +  20  ) * 10.275 + SEL( PLC_PRG.test[91] > 20 , 0.5, -0.5)
  rectangle at (227,214)-(228,224): alarm colour if PLC_PRG.test[92] < 0; top (-1.0 *  PLC_PRG.test[92]  +  20  ) * 10.275 + SEL( PLC_PRG.test[92] > 20 , 0.5, -0.5); bottom (-1.0 *  PLC_PRG.test[92]  +  20  ) * 10.275 + SEL( PLC_PRG.test[92] > 20 , 0.5, -0.5)
  rectangle at (229,214)-(230,224): alarm colour if PLC_PRG.test[93] < 0; top (-1.0 *  PLC_PRG.test[93]  +  20  ) * 10.275 + SEL( PLC_PRG.test[93] > 20 , 0.5, -0.5); bottom (-1.0 *  PLC_PRG.test[93]  +  20  ) * 10.275 + SEL( PLC_PRG.test[93] > 20 , 0.5, -0.5)
  rectangle at (231,214)-(232,224): alarm colour if PLC_PRG.test[94] < 0; top (-1.0 *  PLC_PRG.test[94]  +  20  ) * 10.275 + SEL( PLC_PRG.test[94] > 20 , 0.5, -0.5); bottom (-1.0 *  PLC_PRG.test[94]  +  20  ) * 10.275 + SEL( PLC_PRG.test[94] > 20 , 0.5, -0.5)
  rectangle at (233,214)-(234,224): alarm colour if PLC_PRG.test[95] < 0; top (-1.0 *  PLC_PRG.test[95]  +  20  ) * 10.275 + SEL( PLC_PRG.test[95] > 20 , 0.5, -0.5); bottom (-1.0 *  PLC_PRG.test[95]  +  20  ) * 10.275 + SEL( PLC_PRG.test[95] > 20 , 0.5, -0.5)
  rectangle at (235,214)-(236,224): alarm colour if PLC_PRG.test[96] < 0; top (-1.0 *  PLC_PRG.test[96]  +  20  ) * 10.275 + SEL( PLC_PRG.test[96] > 20 , 0.5, -0.5); bottom (-1.0 *  PLC_PRG.test[96]  +  20  ) * 10.275 + SEL( PLC_PRG.test[96] > 20 , 0.5, -0.5)
  rectangle at (237,214)-(238,224): alarm colour if PLC_PRG.test[97] < 0; top (-1.0 *  PLC_PRG.test[97]  +  20  ) * 10.275 + SEL( PLC_PRG.test[97] > 20 , 0.5, -0.5); bottom (-1.0 *  PLC_PRG.test[97]  +  20  ) * 10.275 + SEL( PLC_PRG.test[97] > 20 , 0.5, -0.5)
  rectangle at (239,214)-(240,224): alarm colour if PLC_PRG.test[98] < 0; top (-1.0 *  PLC_PRG.test[98]  +  20  ) * 10.275 + SEL( PLC_PRG.test[98] > 20 , 0.5, -0.5); bottom (-1.0 *  PLC_PRG.test[98]  +  20  ) * 10.275 + SEL( PLC_PRG.test[98] > 20 , 0.5, -0.5)
  rectangle at (241,214)-(242,224): alarm colour if PLC_PRG.test[99] < 0; top (-1.0 *  PLC_PRG.test[99]  +  20  ) * 10.275 + SEL( PLC_PRG.test[99] > 20 , 0.5, -0.5); bottom (-1.0 *  PLC_PRG.test[99]  +  20  ) * 10.275 + SEL( PLC_PRG.test[99] > 20 , 0.5, -0.5)
  rectangle at (243,214)-(244,224): alarm colour if PLC_PRG.test[100] < 0; top (-1.0 *  PLC_PRG.test[100]  +  20  ) * 10.275 + SEL( PLC_PRG.test[100] > 20 , 0.5, -0.5); bottom (-1.0 *  PLC_PRG.test[100]  +  20  ) * 10.275 + SEL( PLC_PRG.test[100] > 20 , 0.5, -0.5)
  rectangle at (245,214)-(246,224): alarm colour if PLC_PRG.test[101] < 0; top (-1.0 *  PLC_PRG.test[101]  +  20  ) * 10.275 + SEL( PLC_PRG.test[101] > 20 , 0.5, -0.5); bottom (-1.0 *  PLC_PRG.test[101]  +  20  ) * 10.275 + SEL( PLC_PRG.test[101] > 20 , 0.5, -0.5)
  rectangle at (247,214)-(248,224): alarm colour if PLC_PRG.test[102] < 0; top (-1.0 *  PLC_PRG.test[102]  +  20  ) * 10.275 + SEL( PLC_PRG.test[102] > 20 , 0.5, -0.5); bottom (-1.0 *  PLC_PRG.test[102]  +  20  ) * 10.275 + SEL( PLC_PRG.test[102] > 20 , 0.5, -0.5)
  rectangle at (249,214)-(250,224): alarm colour if PLC_PRG.test[103] < 0; top (-1.0 *  PLC_PRG.test[103]  +  20  ) * 10.275 + SEL( PLC_PRG.test[103] > 20 , 0.5, -0.5); bottom (-1.0 *  PLC_PRG.test[103]  +  20  ) * 10.275 + SEL( PLC_PRG.test[103] > 20 , 0.5, -0.5)
  rectangle at (251,214)-(252,224): alarm colour if PLC_PRG.test[104] < 0; top (-1.0 *  PLC_PRG.test[104]  +  20  ) * 10.275 + SEL( PLC_PRG.test[104] > 20 , 0.5, -0.5); bottom (-1.0 *  PLC_PRG.test[104]  +  20  ) * 10.275 + SEL( PLC_PRG.test[104] > 20 , 0.5, -0.5)
  rectangle at (253,214)-(254,224): alarm colour if PLC_PRG.test[105] < 0; top (-1.0 *  PLC_PRG.test[105]  +  20  ) * 10.275 + SEL( PLC_PRG.test[105] > 20 , 0.5, -0.5); bottom (-1.0 *  PLC_PRG.test[105]  +  20  ) * 10.275 + SEL( PLC_PRG.test[105] > 20 , 0.5, -0.5)
  rectangle at (255,214)-(256,224): alarm colour if PLC_PRG.test[106] < 0; top (-1.0 *  PLC_PRG.test[106]  +  20  ) * 10.275 + SEL( PLC_PRG.test[106] > 20 , 0.5, -0.5); bottom (-1.0 *  PLC_PRG.test[106]  +  20  ) * 10.275 + SEL( PLC_PRG.test[106] > 20 , 0.5, -0.5)
  rectangle at (257,214)-(258,224): alarm colour if PLC_PRG.test[107] < 0; top (-1.0 *  PLC_PRG.test[107]  +  20  ) * 10.275 + SEL( PLC_PRG.test[107] > 20 , 0.5, -0.5); bottom (-1.0 *  PLC_PRG.test[107]  +  20  ) * 10.275 + SEL( PLC_PRG.test[107] > 20 , 0.5, -0.5)
  rectangle at (259,214)-(260,224): alarm colour if PLC_PRG.test[108] < 0; top (-1.0 *  PLC_PRG.test[108]  +  20  ) * 10.275 + SEL( PLC_PRG.test[108] > 20 , 0.5, -0.5); bottom (-1.0 *  PLC_PRG.test[108]  +  20  ) * 10.275 + SEL( PLC_PRG.test[108] > 20 , 0.5, -0.5)
  rectangle at (261,214)-(262,224): alarm colour if PLC_PRG.test[109] < 0; top (-1.0 *  PLC_PRG.test[109]  +  20  ) * 10.275 + SEL( PLC_PRG.test[109] > 20 , 0.5, -0.5); bottom (-1.0 *  PLC_PRG.test[109]  +  20  ) * 10.275 + SEL( PLC_PRG.test[109] > 20 , 0.5, -0.5)
  rectangle at (263,214)-(264,224): alarm colour if PLC_PRG.test[110] < 0; top (-1.0 *  PLC_PRG.test[110]  +  20  ) * 10.275 + SEL( PLC_PRG.test[110] > 20 , 0.5, -0.5); bottom (-1.0 *  PLC_PRG.test[110]  +  20  ) * 10.275 + SEL( PLC_PRG.test[110] > 20 , 0.5, -0.5)
  rectangle at (265,214)-(266,224): alarm colour if PLC_PRG.test[111] < 0; top (-1.0 *  PLC_PRG.test[111]  +  20  ) * 10.275 + SEL( PLC_PRG.test[111] > 20 , 0.5, -0.5); bottom (-1.0 *  PLC_PRG.test[111]  +  20  ) * 10.275 + SEL( PLC_PRG.test[111] > 20 , 0.5, -0.5)
  rectangle at (267,214)-(268,224): alarm colour if PLC_PRG.test[112] < 0; top (-1.0 *  PLC_PRG.test[112]  +  20  ) * 10.275 + SEL( PLC_PRG.test[112] > 20 , 0.5, -0.5); bottom (-1.0 *  PLC_PRG.test[112]  +  20  ) * 10.275 + SEL( PLC_PRG.test[112] > 20 , 0.5, -0.5)
  rectangle at (269,214)-(270,224): alarm colour if PLC_PRG.test[113] < 0; top (-1.0 *  PLC_PRG.test[113]  +  20  ) * 10.275 + SEL( PLC_PRG.test[113] > 20 , 0.5, -0.5); bottom (-1.0 *  PLC_PRG.test[113]  +  20  ) * 10.275 + SEL( PLC_PRG.test[113] > 20 , 0.5, -0.5)
  rectangle at (271,214)-(272,224): alarm colour if PLC_PRG.test[114] < 0; top (-1.0 *  PLC_PRG.test[114]  +  20  ) * 10.275 + SEL( PLC_PRG.test[114] > 20 , 0.5, -0.5); bottom (-1.0 *  PLC_PRG.test[114]  +  20  ) * 10.275 + SEL( PLC_PRG.test[114] > 20 , 0.5, -0.5)
  rectangle at (273,214)-(274,224): alarm colour if PLC_PRG.test[115] < 0; top (-1.0 *  PLC_PRG.test[115]  +  20  ) * 10.275 + SEL( PLC_PRG.test[115] > 20 , 0.5, -0.5); bottom (-1.0 *  PLC_PRG.test[115]  +  20  ) * 10.275 + SEL( PLC_PRG.test[115] > 20 , 0.5, -0.5)
  rectangle at (275,214)-(276,224): alarm colour if PLC_PRG.test[116] < 0; top (-1.0 *  PLC_PRG.test[116]  +  20  ) * 10.275 + SEL( PLC_PRG.test[116] > 20 , 0.5, -0.5); bottom (-1.0 *  PLC_PRG.test[116]  +  20  ) * 10.275 + SEL( PLC_PRG.test[116] > 20 , 0.5, -0.5)
  rectangle at (277,214)-(278,224): alarm colour if PLC_PRG.test[117] < 0; top (-1.0 *  PLC_PRG.test[117]  +  20  ) * 10.275 + SEL( PLC_PRG.test[117] > 20 , 0.5, -0.5); bottom (-1.0 *  PLC_PRG.test[117]  +  20  ) * 10.275 + SEL( PLC_PRG.test[117] > 20 , 0.5, -0.5)
  rectangle at (279,214)-(280,224): alarm colour if PLC_PRG.test[118] < 0; top (-1.0 *  PLC_PRG.test[118]  +  20  ) * 10.275 + SEL( PLC_PRG.test[118] > 20 , 0.5, -0.5); bottom (-1.0 *  PLC_PRG.test[118]  +  20  ) * 10.275 + SEL( PLC_PRG.test[118] > 20 , 0.5, -0.5)
  rectangle at (281,214)-(282,224): alarm colour if PLC_PRG.test[119] < 0; top (-1.0 *  PLC_PRG.test[119]  +  20  ) * 10.275 + SEL( PLC_PRG.test[119] > 20 , 0.5, -0.5); bottom (-1.0 *  PLC_PRG.test[119]  +  20  ) * 10.275 + SEL( PLC_PRG.test[119] > 20 , 0.5, -0.5)
  rectangle at (283,214)-(284,224): alarm colour if PLC_PRG.test[120] < 0; top (-1.0 *  PLC_PRG.test[120]  +  20  ) * 10.275 + SEL( PLC_PRG.test[120] > 20 , 0.5, -0.5); bottom (-1.0 *  PLC_PRG.test[120]  +  20  ) * 10.275 + SEL( PLC_PRG.test[120] > 20 , 0.5, -0.5)
  rectangle at (285,214)-(286,224): alarm colour if PLC_PRG.test[121] < 0; top (-1.0 *  PLC_PRG.test[121]  +  20  ) * 10.275 + SEL( PLC_PRG.test[121] > 20 , 0.5, -0.5); bottom (-1.0 *  PLC_PRG.test[121]  +  20  ) * 10.275 + SEL( PLC_PRG.test[121] > 20 , 0.5, -0.5)
  rectangle at (287,214)-(288,224): alarm colour if PLC_PRG.test[122] < 0; top (-1.0 *  PLC_PRG.test[122]  +  20  ) * 10.275 + SEL( PLC_PRG.test[122] > 20 , 0.5, -0.5); bottom (-1.0 *  PLC_PRG.test[122]  +  20  ) * 10.275 + SEL( PLC_PRG.test[122] > 20 , 0.5, -0.5)
  rectangle at (289,214)-(290,224): alarm colour if PLC_PRG.test[123] < 0; top (-1.0 *  PLC_PRG.test[123]  +  20  ) * 10.275 + SEL( PLC_PRG.test[123] > 20 , 0.5, -0.5); bottom (-1.0 *  PLC_PRG.test[123]  +  20  ) * 10.275 + SEL( PLC_PRG.test[123] > 20 , 0.5, -0.5)
  rectangle at (291,214)-(292,224): alarm colour if PLC_PRG.test[124] < 0; top (-1.0 *  PLC_PRG.test[124]  +  20  ) * 10.275 + SEL( PLC_PRG.test[124] > 20 , 0.5, -0.5); bottom (-1.0 *  PLC_PRG.test[124]  +  20  ) * 10.275 + SEL( PLC_PRG.test[124] > 20 , 0.5, -0.5)
  rectangle at (293,214)-(294,224): alarm colour if PLC_PRG.test[125] < 0; top (-1.0 *  PLC_PRG.test[125]  +  20  ) * 10.275 + SEL( PLC_PRG.test[125] > 20 , 0.5, -0.5); bottom (-1.0 *  PLC_PRG.test[125]  +  20  ) * 10.275 + SEL( PLC_PRG.test[125] > 20 , 0.5, -0.5)
  rectangle at (295,214)-(296,224): alarm colour if PLC_PRG.test[126] < 0; top (-1.0 *  PLC_PRG.test[126]  +  20  ) * 10.275 + SEL( PLC_PRG.test[126] > 20 , 0.5, -0.5); bottom (-1.0 *  PLC_PRG.test[126]  +  20  ) * 10.275 + SEL( PLC_PRG.test[126] > 20 , 0.5, -0.5)
  rectangle at (297,214)-(298,224): alarm colour if PLC_PRG.test[127] < 0; top (-1.0 *  PLC_PRG.test[127]  +  20  ) * 10.275 + SEL( PLC_PRG.test[127] > 20 , 0.5, -0.5); bottom (-1.0 *  PLC_PRG.test[127]  +  20  ) * 10.275 + SEL( PLC_PRG.test[127] > 20 , 0.5, -0.5)
  rectangle at (299,214)-(300,224): alarm colour if PLC_PRG.test[128] < 0; top (-1.0 *  PLC_PRG.test[128]  +  20  ) * 10.275 + SEL( PLC_PRG.test[128] > 20 , 0.5, -0.5); bottom (-1.0 *  PLC_PRG.test[128]  +  20  ) * 10.275 + SEL( PLC_PRG.test[128] > 20 , 0.5, -0.5)
  rectangle at (301,214)-(302,224): alarm colour if PLC_PRG.test[129] < 0; top (-1.0 *  PLC_PRG.test[129]  +  20  ) * 10.275 + SEL( PLC_PRG.test[129] > 20 , 0.5, -0.5); bottom (-1.0 *  PLC_PRG.test[129]  +  20  ) * 10.275 + SEL( PLC_PRG.test[129] > 20 , 0.5, -0.5)
  rectangle at (303,214)-(304,224): alarm colour if PLC_PRG.test[130] < 0; top (-1.0 *  PLC_PRG.test[130]  +  20  ) * 10.275 + SEL( PLC_PRG.test[130] > 20 , 0.5, -0.5); bottom (-1.0 *  PLC_PRG.test[130]  +  20  ) * 10.275 + SEL( PLC_PRG.test[130] > 20 , 0.5, -0.5)
  rectangle at (305,214)-(306,224): alarm colour if PLC_PRG.test[131] < 0; top (-1.0 *  PLC_PRG.test[131]  +  20  ) * 10.275 + SEL( PLC_PRG.test[131] > 20 , 0.5, -0.5); bottom (-1.0 *  PLC_PRG.test[131]  +  20  ) * 10.275 + SEL( PLC_PRG.test[131] > 20 , 0.5, -0.5)
  rectangle at (307,214)-(308,224): alarm colour if PLC_PRG.test[132] < 0; top (-1.0 *  PLC_PRG.test[132]  +  20  ) * 10.275 + SEL( PLC_PRG.test[132] > 20 , 0.5, -0.5); bottom (-1.0 *  PLC_PRG.test[132]  +  20  ) * 10.275 + SEL( PLC_PRG.test[132] > 20 , 0.5, -0.5)
  rectangle at (309,214)-(310,224): alarm colour if PLC_PRG.test[133] < 0; top (-1.0 *  PLC_PRG.test[133]  +  20  ) * 10.275 + SEL( PLC_PRG.test[133] > 20 , 0.5, -0.5); bottom (-1.0 *  PLC_PRG.test[133]  +  20  ) * 10.275 + SEL( PLC_PRG.test[133] > 20 , 0.5, -0.5)
  rectangle at (311,214)-(312,224): alarm colour if PLC_PRG.test[134] < 0; top (-1.0 *  PLC_PRG.test[134]  +  20  ) * 10.275 + SEL( PLC_PRG.test[134] > 20 , 0.5, -0.5); bottom (-1.0 *  PLC_PRG.test[134]  +  20  ) * 10.275 + SEL( PLC_PRG.test[134] > 20 , 0.5, -0.5)
  rectangle at (313,214)-(314,224): alarm colour if PLC_PRG.test[135] < 0; top (-1.0 *  PLC_PRG.test[135]  +  20  ) * 10.275 + SEL( PLC_PRG.test[135] > 20 , 0.5, -0.5); bottom (-1.0 *  PLC_PRG.test[135]  +  20  ) * 10.275 + SEL( PLC_PRG.test[135] > 20 , 0.5, -0.5)
  rectangle at (315,214)-(316,224): alarm colour if PLC_PRG.test[136] < 0; top (-1.0 *  PLC_PRG.test[136]  +  20  ) * 10.275 + SEL( PLC_PRG.test[136] > 20 , 0.5, -0.5); bottom (-1.0 *  PLC_PRG.test[136]  +  20  ) * 10.275 + SEL( PLC_PRG.test[136] > 20 , 0.5, -0.5)
  rectangle at (317,214)-(318,224): alarm colour if PLC_PRG.test[137] < 0; top (-1.0 *  PLC_PRG.test[137]  +  20  ) * 10.275 + SEL( PLC_PRG.test[137] > 20 , 0.5, -0.5); bottom (-1.0 *  PLC_PRG.test[137]  +  20  ) * 10.275 + SEL( PLC_PRG.test[137] > 20 , 0.5, -0.5)
  rectangle at (319,214)-(320,224): alarm colour if PLC_PRG.test[138] < 0; top (-1.0 *  PLC_PRG.test[138]  +  20  ) * 10.275 + SEL( PLC_PRG.test[138] > 20 , 0.5, -0.5); bottom (-1.0 *  PLC_PRG.test[138]  +  20  ) * 10.275 + SEL( PLC_PRG.test[138] > 20 , 0.5, -0.5)
  rectangle at (321,214)-(322,224): alarm colour if PLC_PRG.test[139] < 0; top (-1.0 *  PLC_PRG.test[139]  +  20  ) * 10.275 + SEL( PLC_PRG.test[139] > 20 , 0.5, -0.5); bottom (-1.0 *  PLC_PRG.test[139]  +  20  ) * 10.275 + SEL( PLC_PRG.test[139] > 20 , 0.5, -0.5)
  rectangle at (323,214)-(324,224): alarm colour if PLC_PRG.test[140] < 0; top (-1.0 *  PLC_PRG.test[140]  +  20  ) * 10.275 + SEL( PLC_PRG.test[140] > 20 , 0.5, -0.5); bottom (-1.0 *  PLC_PRG.test[140]  +  20  ) * 10.275 + SEL( PLC_PRG.test[140] > 20 , 0.5, -0.5)
  rectangle at (325,214)-(326,224): alarm colour if PLC_PRG.test[141] < 0; top (-1.0 *  PLC_PRG.test[141]  +  20  ) * 10.275 + SEL( PLC_PRG.test[141] > 20 , 0.5, -0.5); bottom (-1.0 *  PLC_PRG.test[141]  +  20  ) * 10.275 + SEL( PLC_PRG.test[141] > 20 , 0.5, -0.5)
  rectangle at (327,214)-(328,224): alarm colour if PLC_PRG.test[142] < 0; top (-1.0 *  PLC_PRG.test[142]  +  20  ) * 10.275 + SEL( PLC_PRG.test[142] > 20 , 0.5, -0.5); bottom (-1.0 *  PLC_PRG.test[142]  +  20  ) * 10.275 + SEL( PLC_PRG.test[142] > 20 , 0.5, -0.5)
  rectangle at (329,214)-(330,224): alarm colour if PLC_PRG.test[143] < 0; top (-1.0 *  PLC_PRG.test[143]  +  20  ) * 10.275 + SEL( PLC_PRG.test[143] > 20 , 0.5, -0.5); bottom (-1.0 *  PLC_PRG.test[143]  +  20  ) * 10.275 + SEL( PLC_PRG.test[143] > 20 , 0.5, -0.5)
  rectangle at (331,214)-(332,224): alarm colour if PLC_PRG.test[144] < 0; top (-1.0 *  PLC_PRG.test[144]  +  20  ) * 10.275 + SEL( PLC_PRG.test[144] > 20 , 0.5, -0.5); bottom (-1.0 *  PLC_PRG.test[144]  +  20  ) * 10.275 + SEL( PLC_PRG.test[144] > 20 , 0.5, -0.5)
  rectangle at (333,214)-(334,224): alarm colour if PLC_PRG.test[145] < 0; top (-1.0 *  PLC_PRG.test[145]  +  20  ) * 10.275 + SEL( PLC_PRG.test[145] > 20 , 0.5, -0.5); bottom (-1.0 *  PLC_PRG.test[145]  +  20  ) * 10.275 + SEL( PLC_PRG.test[145] > 20 , 0.5, -0.5)
  rectangle at (335,214)-(336,224): alarm colour if PLC_PRG.test[146] < 0; top (-1.0 *  PLC_PRG.test[146]  +  20  ) * 10.275 + SEL( PLC_PRG.test[146] > 20 , 0.5, -0.5); bottom (-1.0 *  PLC_PRG.test[146]  +  20  ) * 10.275 + SEL( PLC_PRG.test[146] > 20 , 0.5, -0.5)
  rectangle at (337,214)-(338,224): alarm colour if PLC_PRG.test[147] < 0; top (-1.0 *  PLC_PRG.test[147]  +  20  ) * 10.275 + SEL( PLC_PRG.test[147] > 20 , 0.5, -0.5); bottom (-1.0 *  PLC_PRG.test[147]  +  20  ) * 10.275 + SEL( PLC_PRG.test[147] > 20 , 0.5, -0.5)
  rectangle at (339,214)-(340,224): alarm colour if PLC_PRG.test[148] < 0; top (-1.0 *  PLC_PRG.test[148]  +  20  ) * 10.275 + SEL( PLC_PRG.test[148] > 20 , 0.5, -0.5); bottom (-1.0 *  PLC_PRG.test[148]  +  20  ) * 10.275 + SEL( PLC_PRG.test[148] > 20 , 0.5, -0.5)
  rectangle at (341,214)-(342,224): alarm colour if PLC_PRG.test[149] < 0; top (-1.0 *  PLC_PRG.test[149]  +  20  ) * 10.275 + SEL( PLC_PRG.test[149] > 20 , 0.5, -0.5); bottom (-1.0 *  PLC_PRG.test[149]  +  20  ) * 10.275 + SEL( PLC_PRG.test[149] > 20 , 0.5, -0.5)
  rectangle at (343,214)-(344,224): alarm colour if PLC_PRG.test[150] < 0; top (-1.0 *  PLC_PRG.test[150]  +  20  ) * 10.275 + SEL( PLC_PRG.test[150] > 20 , 0.5, -0.5); bottom (-1.0 *  PLC_PRG.test[150]  +  20  ) * 10.275 + SEL( PLC_PRG.test[150] > 20 , 0.5, -0.5)
  rectangle at (345,214)-(346,224): alarm colour if PLC_PRG.test[151] < 0; top (-1.0 *  PLC_PRG.test[151]  +  20  ) * 10.275 + SEL( PLC_PRG.test[151] > 20 , 0.5, -0.5); bottom (-1.0 *  PLC_PRG.test[151]  +  20  ) * 10.275 + SEL( PLC_PRG.test[151] > 20 , 0.5, -0.5)
  rectangle at (347,214)-(348,224): alarm colour if PLC_PRG.test[152] < 0; top (-1.0 *  PLC_PRG.test[152]  +  20  ) * 10.275 + SEL( PLC_PRG.test[152] > 20 , 0.5, -0.5); bottom (-1.0 *  PLC_PRG.test[152]  +  20  ) * 10.275 + SEL( PLC_PRG.test[152] > 20 , 0.5, -0.5)
  rectangle at (349,214)-(350,224): alarm colour if PLC_PRG.test[153] < 0; top (-1.0 *  PLC_PRG.test[153]  +  20  ) * 10.275 + SEL( PLC_PRG.test[153] > 20 , 0.5, -0.5); bottom (-1.0 *  PLC_PRG.test[153]  +  20  ) * 10.275 + SEL( PLC_PRG.test[153] > 20 , 0.5, -0.5)
  rectangle at (351,214)-(352,224): alarm colour if PLC_PRG.test[154] < 0; top (-1.0 *  PLC_PRG.test[154]  +  20  ) * 10.275 + SEL( PLC_PRG.test[154] > 20 , 0.5, -0.5); bottom (-1.0 *  PLC_PRG.test[154]  +  20  ) * 10.275 + SEL( PLC_PRG.test[154] > 20 , 0.5, -0.5)
  rectangle at (353,214)-(354,224): alarm colour if PLC_PRG.test[155] < 0; top (-1.0 *  PLC_PRG.test[155]  +  20  ) * 10.275 + SEL( PLC_PRG.test[155] > 20 , 0.5, -0.5); bottom (-1.0 *  PLC_PRG.test[155]  +  20  ) * 10.275 + SEL( PLC_PRG.test[155] > 20 , 0.5, -0.5)
  rectangle at (355,214)-(356,224): alarm colour if PLC_PRG.test[156] < 0; top (-1.0 *  PLC_PRG.test[156]  +  20  ) * 10.275 + SEL( PLC_PRG.test[156] > 20 , 0.5, -0.5); bottom (-1.0 *  PLC_PRG.test[156]  +  20  ) * 10.275 + SEL( PLC_PRG.test[156] > 20 , 0.5, -0.5)
  rectangle at (357,214)-(358,224): alarm colour if PLC_PRG.test[157] < 0; top (-1.0 *  PLC_PRG.test[157]  +  20  ) * 10.275 + SEL( PLC_PRG.test[157] > 20 , 0.5, -0.5); bottom (-1.0 *  PLC_PRG.test[157]  +  20  ) * 10.275 + SEL( PLC_PRG.test[157] > 20 , 0.5, -0.5)
  rectangle at (359,214)-(360,224): alarm colour if PLC_PRG.test[158] < 0; top (-1.0 *  PLC_PRG.test[158]  +  20  ) * 10.275 + SEL( PLC_PRG.test[158] > 20 , 0.5, -0.5); bottom (-1.0 *  PLC_PRG.test[158]  +  20  ) * 10.275 + SEL( PLC_PRG.test[158] > 20 , 0.5, -0.5)
  rectangle at (361,214)-(362,224): alarm colour if PLC_PRG.test[159] < 0; top (-1.0 *  PLC_PRG.test[159]  +  20  ) * 10.275 + SEL( PLC_PRG.test[159] > 20 , 0.5, -0.5); bottom (-1.0 *  PLC_PRG.test[159]  +  20  ) * 10.275 + SEL( PLC_PRG.test[159] > 20 , 0.5, -0.5)
  rectangle at (363,214)-(364,224): alarm colour if PLC_PRG.test[160] < 0; top (-1.0 *  PLC_PRG.test[160]  +  20  ) * 10.275 + SEL( PLC_PRG.test[160] > 20 , 0.5, -0.5); bottom (-1.0 *  PLC_PRG.test[160]  +  20  ) * 10.275 + SEL( PLC_PRG.test[160] > 20 , 0.5, -0.5)
  rectangle at (365,214)-(366,224): alarm colour if PLC_PRG.test[161] < 0; top (-1.0 *  PLC_PRG.test[161]  +  20  ) * 10.275 + SEL( PLC_PRG.test[161] > 20 , 0.5, -0.5); bottom (-1.0 *  PLC_PRG.test[161]  +  20  ) * 10.275 + SEL( PLC_PRG.test[161] > 20 , 0.5, -0.5)
  rectangle at (367,214)-(368,224): alarm colour if PLC_PRG.test[162] < 0; top (-1.0 *  PLC_PRG.test[162]  +  20  ) * 10.275 + SEL( PLC_PRG.test[162] > 20 , 0.5, -0.5); bottom (-1.0 *  PLC_PRG.test[162]  +  20  ) * 10.275 + SEL( PLC_PRG.test[162] > 20 , 0.5, -0.5)
  rectangle at (369,214)-(370,224): alarm colour if PLC_PRG.test[163] < 0; top (-1.0 *  PLC_PRG.test[163]  +  20  ) * 10.275 + SEL( PLC_PRG.test[163] > 20 , 0.5, -0.5); bottom (-1.0 *  PLC_PRG.test[163]  +  20  ) * 10.275 + SEL( PLC_PRG.test[163] > 20 , 0.5, -0.5)
  rectangle at (371,214)-(372,224): alarm colour if PLC_PRG.test[164] < 0; top (-1.0 *  PLC_PRG.test[164]  +  20  ) * 10.275 + SEL( PLC_PRG.test[164] > 20 , 0.5, -0.5); bottom (-1.0 *  PLC_PRG.test[164]  +  20  ) * 10.275 + SEL( PLC_PRG.test[164] > 20 , 0.5, -0.5)
  rectangle at (373,214)-(374,224): alarm colour if PLC_PRG.test[165] < 0; top (-1.0 *  PLC_PRG.test[165]  +  20  ) * 10.275 + SEL( PLC_PRG.test[165] > 20 , 0.5, -0.5); bottom (-1.0 *  PLC_PRG.test[165]  +  20  ) * 10.275 + SEL( PLC_PRG.test[165] > 20 , 0.5, -0.5)
  rectangle at (375,214)-(376,224): alarm colour if PLC_PRG.test[166] < 0; top (-1.0 *  PLC_PRG.test[166]  +  20  ) * 10.275 + SEL( PLC_PRG.test[166] > 20 , 0.5, -0.5); bottom (-1.0 *  PLC_PRG.test[166]  +  20  ) * 10.275 + SEL( PLC_PRG.test[166] > 20 , 0.5, -0.5)
  rectangle at (377,214)-(378,224): alarm colour if PLC_PRG.test[167] < 0; top (-1.0 *  PLC_PRG.test[167]  +  20  ) * 10.275 + SEL( PLC_PRG.test[167] > 20 , 0.5, -0.5); bottom (-1.0 *  PLC_PRG.test[167]  +  20  ) * 10.275 + SEL( PLC_PRG.test[167] > 20 , 0.5, -0.5)
  rectangle at (379,214)-(380,224): alarm colour if PLC_PRG.test[168] < 0; top (-1.0 *  PLC_PRG.test[168]  +  20  ) * 10.275 + SEL( PLC_PRG.test[168] > 20 , 0.5, -0.5); bottom (-1.0 *  PLC_PRG.test[168]  +  20  ) * 10.275 + SEL( PLC_PRG.test[168] > 20 , 0.5, -0.5)
  rectangle at (381,214)-(382,224): alarm colour if PLC_PRG.test[169] < 0; top (-1.0 *  PLC_PRG.test[169]  +  20  ) * 10.275 + SEL( PLC_PRG.test[169] > 20 , 0.5, -0.5); bottom (-1.0 *  PLC_PRG.test[169]  +  20  ) * 10.275 + SEL( PLC_PRG.test[169] > 20 , 0.5, -0.5)
  rectangle at (383,214)-(384,224): alarm colour if PLC_PRG.test[170] < 0; top (-1.0 *  PLC_PRG.test[170]  +  20  ) * 10.275 + SEL( PLC_PRG.test[170] > 20 , 0.5, -0.5); bottom (-1.0 *  PLC_PRG.test[170]  +  20  ) * 10.275 + SEL( PLC_PRG.test[170] > 20 , 0.5, -0.5)
  rectangle at (385,214)-(386,224): alarm colour if PLC_PRG.test[171] < 0; top (-1.0 *  PLC_PRG.test[171]  +  20  ) * 10.275 + SEL( PLC_PRG.test[171] > 20 , 0.5, -0.5); bottom (-1.0 *  PLC_PRG.test[171]  +  20  ) * 10.275 + SEL( PLC_PRG.test[171] > 20 , 0.5, -0.5)
  rectangle at (387,214)-(388,224): alarm colour if PLC_PRG.test[172] < 0; top (-1.0 *  PLC_PRG.test[172]  +  20  ) * 10.275 + SEL( PLC_PRG.test[172] > 20 , 0.5, -0.5); bottom (-1.0 *  PLC_PRG.test[172]  +  20  ) * 10.275 + SEL( PLC_PRG.test[172] > 20 , 0.5, -0.5)
  rectangle at (389,214)-(390,224): alarm colour if PLC_PRG.test[173] < 0; top (-1.0 *  PLC_PRG.test[173]  +  20  ) * 10.275 + SEL( PLC_PRG.test[173] > 20 , 0.5, -0.5); bottom (-1.0 *  PLC_PRG.test[173]  +  20  ) * 10.275 + SEL( PLC_PRG.test[173] > 20 , 0.5, -0.5)
  rectangle at (391,214)-(392,224): alarm colour if PLC_PRG.test[174] < 0; top (-1.0 *  PLC_PRG.test[174]  +  20  ) * 10.275 + SEL( PLC_PRG.test[174] > 20 , 0.5, -0.5); bottom (-1.0 *  PLC_PRG.test[174]  +  20  ) * 10.275 + SEL( PLC_PRG.test[174] > 20 , 0.5, -0.5)
  rectangle at (393,214)-(394,224): alarm colour if PLC_PRG.test[175] < 0; top (-1.0 *  PLC_PRG.test[175]  +  20  ) * 10.275 + SEL( PLC_PRG.test[175] > 20 , 0.5, -0.5); bottom (-1.0 *  PLC_PRG.test[175]  +  20  ) * 10.275 + SEL( PLC_PRG.test[175] > 20 , 0.5, -0.5)
  rectangle at (395,214)-(396,224): alarm colour if PLC_PRG.test[176] < 0; top (-1.0 *  PLC_PRG.test[176]  +  20  ) * 10.275 + SEL( PLC_PRG.test[176] > 20 , 0.5, -0.5); bottom (-1.0 *  PLC_PRG.test[176]  +  20  ) * 10.275 + SEL( PLC_PRG.test[176] > 20 , 0.5, -0.5)
  rectangle at (397,214)-(398,224): alarm colour if PLC_PRG.test[177] < 0; top (-1.0 *  PLC_PRG.test[177]  +  20  ) * 10.275 + SEL( PLC_PRG.test[177] > 20 , 0.5, -0.5); bottom (-1.0 *  PLC_PRG.test[177]  +  20  ) * 10.275 + SEL( PLC_PRG.test[177] > 20 , 0.5, -0.5)
  rectangle at (399,214)-(400,224): alarm colour if PLC_PRG.test[178] < 0; top (-1.0 *  PLC_PRG.test[178]  +  20  ) * 10.275 + SEL( PLC_PRG.test[178] > 20 , 0.5, -0.5); bottom (-1.0 *  PLC_PRG.test[178]  +  20  ) * 10.275 + SEL( PLC_PRG.test[178] > 20 , 0.5, -0.5)
  rectangle at (401,214)-(402,224): alarm colour if PLC_PRG.test[179] < 0; top (-1.0 *  PLC_PRG.test[179]  +  20  ) * 10.275 + SEL( PLC_PRG.test[179] > 20 , 0.5, -0.5); bottom (-1.0 *  PLC_PRG.test[179]  +  20  ) * 10.275 + SEL( PLC_PRG.test[179] > 20 , 0.5, -0.5)
  rectangle at (403,214)-(404,224): alarm colour if PLC_PRG.test[180] < 0; top (-1.0 *  PLC_PRG.test[180]  +  20  ) * 10.275 + SEL( PLC_PRG.test[180] > 20 , 0.5, -0.5); bottom (-1.0 *  PLC_PRG.test[180]  +  20  ) * 10.275 + SEL( PLC_PRG.test[180] > 20 , 0.5, -0.5)
  rectangle at (405,214)-(406,224): alarm colour if PLC_PRG.test[181] < 0; top (-1.0 *  PLC_PRG.test[181]  +  20  ) * 10.275 + SEL( PLC_PRG.test[181] > 20 , 0.5, -0.5); bottom (-1.0 *  PLC_PRG.test[181]  +  20  ) * 10.275 + SEL( PLC_PRG.test[181] > 20 , 0.5, -0.5)
  rectangle at (407,214)-(408,224): alarm colour if PLC_PRG.test[182] < 0; top (-1.0 *  PLC_PRG.test[182]  +  20  ) * 10.275 + SEL( PLC_PRG.test[182] > 20 , 0.5, -0.5); bottom (-1.0 *  PLC_PRG.test[182]  +  20  ) * 10.275 + SEL( PLC_PRG.test[182] > 20 , 0.5, -0.5)
  rectangle at (409,214)-(410,224): alarm colour if PLC_PRG.test[183] < 0; top (-1.0 *  PLC_PRG.test[183]  +  20  ) * 10.275 + SEL( PLC_PRG.test[183] > 20 , 0.5, -0.5); bottom (-1.0 *  PLC_PRG.test[183]  +  20  ) * 10.275 + SEL( PLC_PRG.test[183] > 20 , 0.5, -0.5)
  rectangle at (411,214)-(412,224): alarm colour if PLC_PRG.test[184] < 0; top (-1.0 *  PLC_PRG.test[184]  +  20  ) * 10.275 + SEL( PLC_PRG.test[184] > 20 , 0.5, -0.5); bottom (-1.0 *  PLC_PRG.test[184]  +  20  ) * 10.275 + SEL( PLC_PRG.test[184] > 20 , 0.5, -0.5)
  rectangle at (413,214)-(414,224): alarm colour if PLC_PRG.test[185] < 0; top (-1.0 *  PLC_PRG.test[185]  +  20  ) * 10.275 + SEL( PLC_PRG.test[185] > 20 , 0.5, -0.5); bottom (-1.0 *  PLC_PRG.test[185]  +  20  ) * 10.275 + SEL( PLC_PRG.test[185] > 20 , 0.5, -0.5)
  rectangle at (415,214)-(416,224): alarm colour if PLC_PRG.test[186] < 0; top (-1.0 *  PLC_PRG.test[186]  +  20  ) * 10.275 + SEL( PLC_PRG.test[186] > 20 , 0.5, -0.5); bottom (-1.0 *  PLC_PRG.test[186]  +  20  ) * 10.275 + SEL( PLC_PRG.test[186] > 20 , 0.5, -0.5)
  rectangle at (417,214)-(418,224): alarm colour if PLC_PRG.test[187] < 0; top (-1.0 *  PLC_PRG.test[187]  +  20  ) * 10.275 + SEL( PLC_PRG.test[187] > 20 , 0.5, -0.5); bottom (-1.0 *  PLC_PRG.test[187]  +  20  ) * 10.275 + SEL( PLC_PRG.test[187] > 20 , 0.5, -0.5)
  rectangle at (419,214)-(420,224): alarm colour if PLC_PRG.test[188] < 0; top (-1.0 *  PLC_PRG.test[188]  +  20  ) * 10.275 + SEL( PLC_PRG.test[188] > 20 , 0.5, -0.5); bottom (-1.0 *  PLC_PRG.test[188]  +  20  ) * 10.275 + SEL( PLC_PRG.test[188] > 20 , 0.5, -0.5)
  rectangle at (421,214)-(422,224): alarm colour if PLC_PRG.test[189] < 0; top (-1.0 *  PLC_PRG.test[189]  +  20  ) * 10.275 + SEL( PLC_PRG.test[189] > 20 , 0.5, -0.5); bottom (-1.0 *  PLC_PRG.test[189]  +  20  ) * 10.275 + SEL( PLC_PRG.test[189] > 20 , 0.5, -0.5)
  rectangle at (423,214)-(424,224): alarm colour if PLC_PRG.test[190] < 0; top (-1.0 *  PLC_PRG.test[190]  +  20  ) * 10.275 + SEL( PLC_PRG.test[190] > 20 , 0.5, -0.5); bottom (-1.0 *  PLC_PRG.test[190]  +  20  ) * 10.275 + SEL( PLC_PRG.test[190] > 20 , 0.5, -0.5)
  rectangle at (425,214)-(426,224): alarm colour if PLC_PRG.test[191] < 0; top (-1.0 *  PLC_PRG.test[191]  +  20  ) * 10.275 + SEL( PLC_PRG.test[191] > 20 , 0.5, -0.5); bottom (-1.0 *  PLC_PRG.test[191]  +  20  ) * 10.275 + SEL( PLC_PRG.test[191] > 20 , 0.5, -0.5)
  rectangle at (427,214)-(428,224): alarm colour if PLC_PRG.test[192] < 0; top (-1.0 *  PLC_PRG.test[192]  +  20  ) * 10.275 + SEL( PLC_PRG.test[192] > 20 , 0.5, -0.5); bottom (-1.0 *  PLC_PRG.test[192]  +  20  ) * 10.275 + SEL( PLC_PRG.test[192] > 20 , 0.5, -0.5)
  rectangle at (429,214)-(430,224): alarm colour if PLC_PRG.test[193] < 0; top (-1.0 *  PLC_PRG.test[193]  +  20  ) * 10.275 + SEL( PLC_PRG.test[193] > 20 , 0.5, -0.5); bottom (-1.0 *  PLC_PRG.test[193]  +  20  ) * 10.275 + SEL( PLC_PRG.test[193] > 20 , 0.5, -0.5)
  rectangle at (431,214)-(432,224): alarm colour if PLC_PRG.test[194] < 0; top (-1.0 *  PLC_PRG.test[194]  +  20  ) * 10.275 + SEL( PLC_PRG.test[194] > 20 , 0.5, -0.5); bottom (-1.0 *  PLC_PRG.test[194]  +  20  ) * 10.275 + SEL( PLC_PRG.test[194] > 20 , 0.5, -0.5)
  rectangle at (433,214)-(434,224): alarm colour if PLC_PRG.test[195] < 0; top (-1.0 *  PLC_PRG.test[195]  +  20  ) * 10.275 + SEL( PLC_PRG.test[195] > 20 , 0.5, -0.5); bottom (-1.0 *  PLC_PRG.test[195]  +  20  ) * 10.275 + SEL( PLC_PRG.test[195] > 20 , 0.5, -0.5)
  rectangle at (435,214)-(436,224): alarm colour if PLC_PRG.test[196] < 0; top (-1.0 *  PLC_PRG.test[196]  +  20  ) * 10.275 + SEL( PLC_PRG.test[196] > 20 , 0.5, -0.5); bottom (-1.0 *  PLC_PRG.test[196]  +  20  ) * 10.275 + SEL( PLC_PRG.test[196] > 20 , 0.5, -0.5)
  rectangle at (437,214)-(438,224): alarm colour if PLC_PRG.test[197] < 0; top (-1.0 *  PLC_PRG.test[197]  +  20  ) * 10.275 + SEL( PLC_PRG.test[197] > 20 , 0.5, -0.5); bottom (-1.0 *  PLC_PRG.test[197]  +  20  ) * 10.275 + SEL( PLC_PRG.test[197] > 20 , 0.5, -0.5)
  rectangle at (439,214)-(440,224): alarm colour if PLC_PRG.test[198] < 0; top (-1.0 *  PLC_PRG.test[198]  +  20  ) * 10.275 + SEL( PLC_PRG.test[198] > 20 , 0.5, -0.5); bottom (-1.0 *  PLC_PRG.test[198]  +  20  ) * 10.275 + SEL( PLC_PRG.test[198] > 20 , 0.5, -0.5)
  rectangle at (441,214)-(442,224): alarm colour if PLC_PRG.test[199] < 0; top (-1.0 *  PLC_PRG.test[199]  +  20  ) * 10.275 + SEL( PLC_PRG.test[199] > 20 , 0.5, -0.5); bottom (-1.0 *  PLC_PRG.test[199]  +  20  ) * 10.275 + SEL( PLC_PRG.test[199] > 20 , 0.5, -0.5)
  rectangle at (443,214)-(444,224): alarm colour if PLC_PRG.test[200] < 0; top (-1.0 *  PLC_PRG.test[200]  +  20  ) * 10.275 + SEL( PLC_PRG.test[200] > 20 , 0.5, -0.5); bottom (-1.0 *  PLC_PRG.test[200]  +  20  ) * 10.275 + SEL( PLC_PRG.test[200] > 20 , 0.5, -0.5)
  rectangle at (445,214)-(446,224): alarm colour if PLC_PRG.test[201] < 0; top (-1.0 *  PLC_PRG.test[201]  +  20  ) * 10.275 + SEL( PLC_PRG.test[201] > 20 , 0.5, -0.5); bottom (-1.0 *  PLC_PRG.test[201]  +  20  ) * 10.275 + SEL( PLC_PRG.test[201] > 20 , 0.5, -0.5)
  rectangle at (447,214)-(448,224): alarm colour if PLC_PRG.test[202] < 0; top (-1.0 *  PLC_PRG.test[202]  +  20  ) * 10.275 + SEL( PLC_PRG.test[202] > 20 , 0.5, -0.5); bottom (-1.0 *  PLC_PRG.test[202]  +  20  ) * 10.275 + SEL( PLC_PRG.test[202] > 20 , 0.5, -0.5)
  rectangle at (449,214)-(450,224): alarm colour if PLC_PRG.test[203] < 0; top (-1.0 *  PLC_PRG.test[203]  +  20  ) * 10.275 + SEL( PLC_PRG.test[203] > 20 , 0.5, -0.5); bottom (-1.0 *  PLC_PRG.test[203]  +  20  ) * 10.275 + SEL( PLC_PRG.test[203] > 20 , 0.5, -0.5)
  rectangle at (451,214)-(452,224): alarm colour if PLC_PRG.test[204] < 0; top (-1.0 *  PLC_PRG.test[204]  +  20  ) * 10.275 + SEL( PLC_PRG.test[204] > 20 , 0.5, -0.5); bottom (-1.0 *  PLC_PRG.test[204]  +  20  ) * 10.275 + SEL( PLC_PRG.test[204] > 20 , 0.5, -0.5)
  rectangle at (453,214)-(454,224): alarm colour if PLC_PRG.test[205] < 0; top (-1.0 *  PLC_PRG.test[205]  +  20  ) * 10.275 + SEL( PLC_PRG.test[205] > 20 , 0.5, -0.5); bottom (-1.0 *  PLC_PRG.test[205]  +  20  ) * 10.275 + SEL( PLC_PRG.test[205] > 20 , 0.5, -0.5)
  rectangle at (455,214)-(456,224): alarm colour if PLC_PRG.test[206] < 0; top (-1.0 *  PLC_PRG.test[206]  +  20  ) * 10.275 + SEL( PLC_PRG.test[206] > 20 , 0.5, -0.5); bottom (-1.0 *  PLC_PRG.test[206]  +  20  ) * 10.275 + SEL( PLC_PRG.test[206] > 20 , 0.5, -0.5)
  rectangle at (457,214)-(458,224): alarm colour if PLC_PRG.test[207] < 0; top (-1.0 *  PLC_PRG.test[207]  +  20  ) * 10.275 + SEL( PLC_PRG.test[207] > 20 , 0.5, -0.5); bottom (-1.0 *  PLC_PRG.test[207]  +  20  ) * 10.275 + SEL( PLC_PRG.test[207] > 20 , 0.5, -0.5)
  rectangle at (459,214)-(460,224): alarm colour if PLC_PRG.test[208] < 0; top (-1.0 *  PLC_PRG.test[208]  +  20  ) * 10.275 + SEL( PLC_PRG.test[208] > 20 , 0.5, -0.5); bottom (-1.0 *  PLC_PRG.test[208]  +  20  ) * 10.275 + SEL( PLC_PRG.test[208] > 20 , 0.5, -0.5)
  rectangle at (461,214)-(462,224): alarm colour if PLC_PRG.test[209] < 0; top (-1.0 *  PLC_PRG.test[209]  +  20  ) * 10.275 + SEL( PLC_PRG.test[209] > 20 , 0.5, -0.5); bottom (-1.0 *  PLC_PRG.test[209]  +  20  ) * 10.275 + SEL( PLC_PRG.test[209] > 20 , 0.5, -0.5)
  rectangle at (463,214)-(464,224): alarm colour if PLC_PRG.test[210] < 0; top (-1.0 *  PLC_PRG.test[210]  +  20  ) * 10.275 + SEL( PLC_PRG.test[210] > 20 , 0.5, -0.5); bottom (-1.0 *  PLC_PRG.test[210]  +  20  ) * 10.275 + SEL( PLC_PRG.test[210] > 20 , 0.5, -0.5)
  rectangle at (465,214)-(466,224): alarm colour if PLC_PRG.test[211] < 0; top (-1.0 *  PLC_PRG.test[211]  +  20  ) * 10.275 + SEL( PLC_PRG.test[211] > 20 , 0.5, -0.5); bottom (-1.0 *  PLC_PRG.test[211]  +  20  ) * 10.275 + SEL( PLC_PRG.test[211] > 20 , 0.5, -0.5)
  rectangle at (467,214)-(468,224): alarm colour if PLC_PRG.test[212] < 0; top (-1.0 *  PLC_PRG.test[212]  +  20  ) * 10.275 + SEL( PLC_PRG.test[212] > 20 , 0.5, -0.5); bottom (-1.0 *  PLC_PRG.test[212]  +  20  ) * 10.275 + SEL( PLC_PRG.test[212] > 20 , 0.5, -0.5)
  rectangle at (469,214)-(470,224): alarm colour if PLC_PRG.test[213] < 0; top (-1.0 *  PLC_PRG.test[213]  +  20  ) * 10.275 + SEL( PLC_PRG.test[213] > 20 , 0.5, -0.5); bottom (-1.0 *  PLC_PRG.test[213]  +  20  ) * 10.275 + SEL( PLC_PRG.test[213] > 20 , 0.5, -0.5)
  rectangle at (471,214)-(472,224): alarm colour if PLC_PRG.test[214] < 0; top (-1.0 *  PLC_PRG.test[214]  +  20  ) * 10.275 + SEL( PLC_PRG.test[214] > 20 , 0.5, -0.5); bottom (-1.0 *  PLC_PRG.test[214]  +  20  ) * 10.275 + SEL( PLC_PRG.test[214] > 20 , 0.5, -0.5)
  rectangle at (473,214)-(474,224): alarm colour if PLC_PRG.test[215] < 0; top (-1.0 *  PLC_PRG.test[215]  +  20  ) * 10.275 + SEL( PLC_PRG.test[215] > 20 , 0.5, -0.5); bottom (-1.0 *  PLC_PRG.test[215]  +  20  ) * 10.275 + SEL( PLC_PRG.test[215] > 20 , 0.5, -0.5)
  rectangle at (475,214)-(476,224): alarm colour if PLC_PRG.test[216] < 0; top (-1.0 *  PLC_PRG.test[216]  +  20  ) * 10.275 + SEL( PLC_PRG.test[216] > 20 , 0.5, -0.5); bottom (-1.0 *  PLC_PRG.test[216]  +  20  ) * 10.275 + SEL( PLC_PRG.test[216] > 20 , 0.5, -0.5)
  rectangle at (477,214)-(478,224): alarm colour if PLC_PRG.test[217] < 0; top (-1.0 *  PLC_PRG.test[217]  +  20  ) * 10.275 + SEL( PLC_PRG.test[217] > 20 , 0.5, -0.5); bottom (-1.0 *  PLC_PRG.test[217]  +  20  ) * 10.275 + SEL( PLC_PRG.test[217] > 20 , 0.5, -0.5)
  rectangle at (479,214)-(480,224): alarm colour if PLC_PRG.test[218] < 0; top (-1.0 *  PLC_PRG.test[218]  +  20  ) * 10.275 + SEL( PLC_PRG.test[218] > 20 , 0.5, -0.5); bottom (-1.0 *  PLC_PRG.test[218]  +  20  ) * 10.275 + SEL( PLC_PRG.test[218] > 20 , 0.5, -0.5)
  rectangle at (481,214)-(482,224): alarm colour if PLC_PRG.test[219] < 0; top (-1.0 *  PLC_PRG.test[219]  +  20  ) * 10.275 + SEL( PLC_PRG.test[219] > 20 , 0.5, -0.5); bottom (-1.0 *  PLC_PRG.test[219]  +  20  ) * 10.275 + SEL( PLC_PRG.test[219] > 20 , 0.5, -0.5)
  rectangle at (483,214)-(484,224): alarm colour if PLC_PRG.test[220] < 0; top (-1.0 *  PLC_PRG.test[220]  +  20  ) * 10.275 + SEL( PLC_PRG.test[220] > 20 , 0.5, -0.5); bottom (-1.0 *  PLC_PRG.test[220]  +  20  ) * 10.275 + SEL( PLC_PRG.test[220] > 20 , 0.5, -0.5)
  rectangle at (485,214)-(486,224): alarm colour if PLC_PRG.test[221] < 0; top (-1.0 *  PLC_PRG.test[221]  +  20  ) * 10.275 + SEL( PLC_PRG.test[221] > 20 , 0.5, -0.5); bottom (-1.0 *  PLC_PRG.test[221]  +  20  ) * 10.275 + SEL( PLC_PRG.test[221] > 20 , 0.5, -0.5)
  rectangle at (487,214)-(488,224): alarm colour if PLC_PRG.test[222] < 0; top (-1.0 *  PLC_PRG.test[222]  +  20  ) * 10.275 + SEL( PLC_PRG.test[222] > 20 , 0.5, -0.5); bottom (-1.0 *  PLC_PRG.test[222]  +  20  ) * 10.275 + SEL( PLC_PRG.test[222] > 20 , 0.5, -0.5)
  rectangle at (489,214)-(490,224): alarm colour if PLC_PRG.test[223] < 0; top (-1.0 *  PLC_PRG.test[223]  +  20  ) * 10.275 + SEL( PLC_PRG.test[223] > 20 , 0.5, -0.5); bottom (-1.0 *  PLC_PRG.test[223]  +  20  ) * 10.275 + SEL( PLC_PRG.test[223] > 20 , 0.5, -0.5)
  rectangle at (491,214)-(492,224): alarm colour if PLC_PRG.test[224] < 0; top (-1.0 *  PLC_PRG.test[224]  +  20  ) * 10.275 + SEL( PLC_PRG.test[224] > 20 , 0.5, -0.5); bottom (-1.0 *  PLC_PRG.test[224]  +  20  ) * 10.275 + SEL( PLC_PRG.test[224] > 20 , 0.5, -0.5)
  rectangle at (493,214)-(494,224): alarm colour if PLC_PRG.test[225] < 0; top (-1.0 *  PLC_PRG.test[225]  +  20  ) * 10.275 + SEL( PLC_PRG.test[225] > 20 , 0.5, -0.5); bottom (-1.0 *  PLC_PRG.test[225]  +  20  ) * 10.275 + SEL( PLC_PRG.test[225] > 20 , 0.5, -0.5)
  rectangle at (495,214)-(496,224): alarm colour if PLC_PRG.test[226] < 0; top (-1.0 *  PLC_PRG.test[226]  +  20  ) * 10.275 + SEL( PLC_PRG.test[226] > 20 , 0.5, -0.5); bottom (-1.0 *  PLC_PRG.test[226]  +  20  ) * 10.275 + SEL( PLC_PRG.test[226] > 20 , 0.5, -0.5)
  rectangle at (497,214)-(498,224): alarm colour if PLC_PRG.test[227] < 0; top (-1.0 *  PLC_PRG.test[227]  +  20  ) * 10.275 + SEL( PLC_PRG.test[227] > 20 , 0.5, -0.5); bottom (-1.0 *  PLC_PRG.test[227]  +  20  ) * 10.275 + SEL( PLC_PRG.test[227] > 20 , 0.5, -0.5)
  rectangle at (499,214)-(500,224): alarm colour if PLC_PRG.test[228] < 0; top (-1.0 *  PLC_PRG.test[228]  +  20  ) * 10.275 + SEL( PLC_PRG.test[228] > 20 , 0.5, -0.5); bottom (-1.0 *  PLC_PRG.test[228]  +  20  ) * 10.275 + SEL( PLC_PRG.test[228] > 20 , 0.5, -0.5)
  rectangle at (501,214)-(502,224): alarm colour if PLC_PRG.test[229] < 0; top (-1.0 *  PLC_PRG.test[229]  +  20  ) * 10.275 + SEL( PLC_PRG.test[229] > 20 , 0.5, -0.5); bottom (-1.0 *  PLC_PRG.test[229]  +  20  ) * 10.275 + SEL( PLC_PRG.test[229] > 20 , 0.5, -0.5)
  rectangle at (503,214)-(504,224): alarm colour if PLC_PRG.test[230] < 0; top (-1.0 *  PLC_PRG.test[230]  +  20  ) * 10.275 + SEL( PLC_PRG.test[230] > 20 , 0.5, -0.5); bottom (-1.0 *  PLC_PRG.test[230]  +  20  ) * 10.275 + SEL( PLC_PRG.test[230] > 20 , 0.5, -0.5)
  rectangle at (505,214)-(506,224): alarm colour if PLC_PRG.test[231] < 0; top (-1.0 *  PLC_PRG.test[231]  +  20  ) * 10.275 + SEL( PLC_PRG.test[231] > 20 , 0.5, -0.5); bottom (-1.0 *  PLC_PRG.test[231]  +  20  ) * 10.275 + SEL( PLC_PRG.test[231] > 20 , 0.5, -0.5)
  rectangle at (507,214)-(508,224): alarm colour if PLC_PRG.test[232] < 0; top (-1.0 *  PLC_PRG.test[232]  +  20  ) * 10.275 + SEL( PLC_PRG.test[232] > 20 , 0.5, -0.5); bottom (-1.0 *  PLC_PRG.test[232]  +  20  ) * 10.275 + SEL( PLC_PRG.test[232] > 20 , 0.5, -0.5)
  rectangle at (509,214)-(510,224): alarm colour if PLC_PRG.test[233] < 0; top (-1.0 *  PLC_PRG.test[233]  +  20  ) * 10.275 + SEL( PLC_PRG.test[233] > 20 , 0.5, -0.5); bottom (-1.0 *  PLC_PRG.test[233]  +  20  ) * 10.275 + SEL( PLC_PRG.test[233] > 20 , 0.5, -0.5)
  rectangle at (511,214)-(512,224): alarm colour if PLC_PRG.test[234] < 0; top (-1.0 *  PLC_PRG.test[234]  +  20  ) * 10.275 + SEL( PLC_PRG.test[234] > 20 , 0.5, -0.5); bottom (-1.0 *  PLC_PRG.test[234]  +  20  ) * 10.275 + SEL( PLC_PRG.test[234] > 20 , 0.5, -0.5)
  rectangle at (513,214)-(514,224): alarm colour if PLC_PRG.test[235] < 0; top (-1.0 *  PLC_PRG.test[235]  +  20  ) * 10.275 + SEL( PLC_PRG.test[235] > 20 , 0.5, -0.5); bottom (-1.0 *  PLC_PRG.test[235]  +  20  ) * 10.275 + SEL( PLC_PRG.test[235] > 20 , 0.5, -0.5)
  rectangle at (515,214)-(516,224): alarm colour if PLC_PRG.test[236] < 0; top (-1.0 *  PLC_PRG.test[236]  +  20  ) * 10.275 + SEL( PLC_PRG.test[236] > 20 , 0.5, -0.5); bottom (-1.0 *  PLC_PRG.test[236]  +  20  ) * 10.275 + SEL( PLC_PRG.test[236] > 20 , 0.5, -0.5)
  rectangle at (517,214)-(518,224): alarm colour if PLC_PRG.test[237] < 0; top (-1.0 *  PLC_PRG.test[237]  +  20  ) * 10.275 + SEL( PLC_PRG.test[237] > 20 , 0.5, -0.5); bottom (-1.0 *  PLC_PRG.test[237]  +  20  ) * 10.275 + SEL( PLC_PRG.test[237] > 20 , 0.5, -0.5)
  rectangle at (519,214)-(520,224): alarm colour if PLC_PRG.test[238] < 0; top (-1.0 *  PLC_PRG.test[238]  +  20  ) * 10.275 + SEL( PLC_PRG.test[238] > 20 , 0.5, -0.5); bottom (-1.0 *  PLC_PRG.test[238]  +  20  ) * 10.275 + SEL( PLC_PRG.test[238] > 20 , 0.5, -0.5)
  rectangle at (521,214)-(522,224): alarm colour if PLC_PRG.test[239] < 0; top (-1.0 *  PLC_PRG.test[239]  +  20  ) * 10.275 + SEL( PLC_PRG.test[239] > 20 , 0.5, -0.5); bottom (-1.0 *  PLC_PRG.test[239]  +  20  ) * 10.275 + SEL( PLC_PRG.test[239] > 20 , 0.5, -0.5)
  rectangle at (523,214)-(524,224): alarm colour if PLC_PRG.test[240] < 0; top (-1.0 *  PLC_PRG.test[240]  +  20  ) * 10.275 + SEL( PLC_PRG.test[240] > 20 , 0.5, -0.5); bottom (-1.0 *  PLC_PRG.test[240]  +  20  ) * 10.275 + SEL( PLC_PRG.test[240] > 20 , 0.5, -0.5)
  rectangle at (525,214)-(526,224): alarm colour if PLC_PRG.test[241] < 0; top (-1.0 *  PLC_PRG.test[241]  +  20  ) * 10.275 + SEL( PLC_PRG.test[241] > 20 , 0.5, -0.5); bottom (-1.0 *  PLC_PRG.test[241]  +  20  ) * 10.275 + SEL( PLC_PRG.test[241] > 20 , 0.5, -0.5)
  rectangle at (527,214)-(528,224): alarm colour if PLC_PRG.test[242] < 0; top (-1.0 *  PLC_PRG.test[242]  +  20  ) * 10.275 + SEL( PLC_PRG.test[242] > 20 , 0.5, -0.5); bottom (-1.0 *  PLC_PRG.test[242]  +  20  ) * 10.275 + SEL( PLC_PRG.test[242] > 20 , 0.5, -0.5)
  rectangle at (529,214)-(530,224): alarm colour if PLC_PRG.test[243] < 0; top (-1.0 *  PLC_PRG.test[243]  +  20  ) * 10.275 + SEL( PLC_PRG.test[243] > 20 , 0.5, -0.5); bottom (-1.0 *  PLC_PRG.test[243]  +  20  ) * 10.275 + SEL( PLC_PRG.test[243] > 20 , 0.5, -0.5)
  rectangle at (531,214)-(532,224): alarm colour if PLC_PRG.test[244] < 0; top (-1.0 *  PLC_PRG.test[244]  +  20  ) * 10.275 + SEL( PLC_PRG.test[244] > 20 , 0.5, -0.5); bottom (-1.0 *  PLC_PRG.test[244]  +  20  ) * 10.275 + SEL( PLC_PRG.test[244] > 20 , 0.5, -0.5)
  rectangle at (533,214)-(534,224): alarm colour if PLC_PRG.test[245] < 0; top (-1.0 *  PLC_PRG.test[245]  +  20  ) * 10.275 + SEL( PLC_PRG.test[245] > 20 , 0.5, -0.5); bottom (-1.0 *  PLC_PRG.test[245]  +  20  ) * 10.275 + SEL( PLC_PRG.test[245] > 20 , 0.5, -0.5)
  rectangle at (535,214)-(536,224): alarm colour if PLC_PRG.test[246] < 0; top (-1.0 *  PLC_PRG.test[246]  +  20  ) * 10.275 + SEL( PLC_PRG.test[246] > 20 , 0.5, -0.5); bottom (-1.0 *  PLC_PRG.test[246]  +  20  ) * 10.275 + SEL( PLC_PRG.test[246] > 20 , 0.5, -0.5)
  rectangle at (537,214)-(538,224): alarm colour if PLC_PRG.test[247] < 0; top (-1.0 *  PLC_PRG.test[247]  +  20  ) * 10.275 + SEL( PLC_PRG.test[247] > 20 , 0.5, -0.5); bottom (-1.0 *  PLC_PRG.test[247]  +  20  ) * 10.275 + SEL( PLC_PRG.test[247] > 20 , 0.5, -0.5)
  rectangle at (539,214)-(540,224): alarm colour if PLC_PRG.test[248] < 0; top (-1.0 *  PLC_PRG.test[248]  +  20  ) * 10.275 + SEL( PLC_PRG.test[248] > 20 , 0.5, -0.5); bottom (-1.0 *  PLC_PRG.test[248]  +  20  ) * 10.275 + SEL( PLC_PRG.test[248] > 20 , 0.5, -0.5)
  rectangle at (541,214)-(542,224): alarm colour if PLC_PRG.test[249] < 0; top (-1.0 *  PLC_PRG.test[249]  +  20  ) * 10.275 + SEL( PLC_PRG.test[249] > 20 , 0.5, -0.5); bottom (-1.0 *  PLC_PRG.test[249]  +  20  ) * 10.275 + SEL( PLC_PRG.test[249] > 20 , 0.5, -0.5)
  rectangle at (543,214)-(544,224): alarm colour if PLC_PRG.test[250] < 0; top (-1.0 *  PLC_PRG.test[250]  +  20  ) * 10.275 + SEL( PLC_PRG.test[250] > 20 , 0.5, -0.5); bottom (-1.0 *  PLC_PRG.test[250]  +  20  ) * 10.275 + SEL( PLC_PRG.test[250] > 20 , 0.5, -0.5)
  rectangle at (545,214)-(546,224): alarm colour if PLC_PRG.test[251] < 0; top (-1.0 *  PLC_PRG.test[251]  +  20  ) * 10.275 + SEL( PLC_PRG.test[251] > 20 , 0.5, -0.5); bottom (-1.0 *  PLC_PRG.test[251]  +  20  ) * 10.275 + SEL( PLC_PRG.test[251] > 20 , 0.5, -0.5)
  rectangle at (547,214)-(548,224): alarm colour if PLC_PRG.test[252] < 0; top (-1.0 *  PLC_PRG.test[252]  +  20  ) * 10.275 + SEL( PLC_PRG.test[252] > 20 , 0.5, -0.5); bottom (-1.0 *  PLC_PRG.test[252]  +  20  ) * 10.275 + SEL( PLC_PRG.test[252] > 20 , 0.5, -0.5)
  rectangle at (549,214)-(550,224): alarm colour if PLC_PRG.test[253] < 0; top (-1.0 *  PLC_PRG.test[253]  +  20  ) * 10.275 + SEL( PLC_PRG.test[253] > 20 , 0.5, -0.5); bottom (-1.0 *  PLC_PRG.test[253]  +  20  ) * 10.275 + SEL( PLC_PRG.test[253] > 20 , 0.5, -0.5)
  rectangle at (551,214)-(552,224): alarm colour if PLC_PRG.test[254] < 0; top (-1.0 *  PLC_PRG.test[254]  +  20  ) * 10.275 + SEL( PLC_PRG.test[254] > 20 , 0.5, -0.5); bottom (-1.0 *  PLC_PRG.test[254]  +  20  ) * 10.275 + SEL( PLC_PRG.test[254] > 20 , 0.5, -0.5)
  rectangle at (553,214)-(554,224): alarm colour if PLC_PRG.test[255] < 0; top (-1.0 *  PLC_PRG.test[255]  +  20  ) * 10.275 + SEL( PLC_PRG.test[255] > 20 , 0.5, -0.5); bottom (-1.0 *  PLC_PRG.test[255]  +  20  ) * 10.275 + SEL( PLC_PRG.test[255] > 20 , 0.5, -0.5)
  rectangle at (555,214)-(556,224): alarm colour if PLC_PRG.test[256] < 0; top (-1.0 *  PLC_PRG.test[256]  +  20  ) * 10.275 + SEL( PLC_PRG.test[256] > 20 , 0.5, -0.5); bottom (-1.0 *  PLC_PRG.test[256]  +  20  ) * 10.275 + SEL( PLC_PRG.test[256] > 20 , 0.5, -0.5)
  rectangle at (557,214)-(558,224): alarm colour if PLC_PRG.test[257] < 0; top (-1.0 *  PLC_PRG.test[257]  +  20  ) * 10.275 + SEL( PLC_PRG.test[257] > 20 , 0.5, -0.5); bottom (-1.0 *  PLC_PRG.test[257]  +  20  ) * 10.275 + SEL( PLC_PRG.test[257] > 20 , 0.5, -0.5)
  rectangle at (559,214)-(560,224): alarm colour if PLC_PRG.test[258] < 0; top (-1.0 *  PLC_PRG.test[258]  +  20  ) * 10.275 + SEL( PLC_PRG.test[258] > 20 , 0.5, -0.5); bottom (-1.0 *  PLC_PRG.test[258]  +  20  ) * 10.275 + SEL( PLC_PRG.test[258] > 20 , 0.5, -0.5)
  rectangle at (561,214)-(562,224): alarm colour if PLC_PRG.test[259] < 0; top (-1.0 *  PLC_PRG.test[259]  +  20  ) * 10.275 + SEL( PLC_PRG.test[259] > 20 , 0.5, -0.5); bottom (-1.0 *  PLC_PRG.test[259]  +  20  ) * 10.275 + SEL( PLC_PRG.test[259] > 20 , 0.5, -0.5)
  rectangle at (563,214)-(564,224): alarm colour if PLC_PRG.test[260] < 0; top (-1.0 *  PLC_PRG.test[260]  +  20  ) * 10.275 + SEL( PLC_PRG.test[260] > 20 , 0.5, -0.5); bottom (-1.0 *  PLC_PRG.test[260]  +  20  ) * 10.275 + SEL( PLC_PRG.test[260] > 20 , 0.5, -0.5)
  rectangle at (565,214)-(566,224): alarm colour if PLC_PRG.test[261] < 0; top (-1.0 *  PLC_PRG.test[261]  +  20  ) * 10.275 + SEL( PLC_PRG.test[261] > 20 , 0.5, -0.5); bottom (-1.0 *  PLC_PRG.test[261]  +  20  ) * 10.275 + SEL( PLC_PRG.test[261] > 20 , 0.5, -0.5)
  rectangle at (567,214)-(568,224): alarm colour if PLC_PRG.test[262] < 0; top (-1.0 *  PLC_PRG.test[262]  +  20  ) * 10.275 + SEL( PLC_PRG.test[262] > 20 , 0.5, -0.5); bottom (-1.0 *  PLC_PRG.test[262]  +  20  ) * 10.275 + SEL( PLC_PRG.test[262] > 20 , 0.5, -0.5)
  rectangle at (569,214)-(570,224): alarm colour if PLC_PRG.test[263] < 0; top (-1.0 *  PLC_PRG.test[263]  +  20  ) * 10.275 + SEL( PLC_PRG.test[263] > 20 , 0.5, -0.5); bottom (-1.0 *  PLC_PRG.test[263]  +  20  ) * 10.275 + SEL( PLC_PRG.test[263] > 20 , 0.5, -0.5)
  rectangle at (571,214)-(572,224): alarm colour if PLC_PRG.test[264] < 0; top (-1.0 *  PLC_PRG.test[264]  +  20  ) * 10.275 + SEL( PLC_PRG.test[264] > 20 , 0.5, -0.5); bottom (-1.0 *  PLC_PRG.test[264]  +  20  ) * 10.275 + SEL( PLC_PRG.test[264] > 20 , 0.5, -0.5)
  rectangle at (573,214)-(574,224): alarm colour if PLC_PRG.test[265] < 0; top (-1.0 *  PLC_PRG.test[265]  +  20  ) * 10.275 + SEL( PLC_PRG.test[265] > 20 , 0.5, -0.5); bottom (-1.0 *  PLC_PRG.test[265]  +  20  ) * 10.275 + SEL( PLC_PRG.test[265] > 20 , 0.5, -0.5)
  rectangle at (575,214)-(576,224): alarm colour if PLC_PRG.test[266] < 0; top (-1.0 *  PLC_PRG.test[266]  +  20  ) * 10.275 + SEL( PLC_PRG.test[266] > 20 , 0.5, -0.5); bottom (-1.0 *  PLC_PRG.test[266]  +  20  ) * 10.275 + SEL( PLC_PRG.test[266] > 20 , 0.5, -0.5)
  rectangle at (577,214)-(578,224): alarm colour if PLC_PRG.test[267] < 0; top (-1.0 *  PLC_PRG.test[267]  +  20  ) * 10.275 + SEL( PLC_PRG.test[267] > 20 , 0.5, -0.5); bottom (-1.0 *  PLC_PRG.test[267]  +  20  ) * 10.275 + SEL( PLC_PRG.test[267] > 20 , 0.5, -0.5)
  rectangle at (579,214)-(580,224): alarm colour if PLC_PRG.test[268] < 0; top (-1.0 *  PLC_PRG.test[268]  +  20  ) * 10.275 + SEL( PLC_PRG.test[268] > 20 , 0.5, -0.5); bottom (-1.0 *  PLC_PRG.test[268]  +  20  ) * 10.275 + SEL( PLC_PRG.test[268] > 20 , 0.5, -0.5)
  rectangle at (581,214)-(582,224): alarm colour if PLC_PRG.test[269] < 0; top (-1.0 *  PLC_PRG.test[269]  +  20  ) * 10.275 + SEL( PLC_PRG.test[269] > 20 , 0.5, -0.5); bottom (-1.0 *  PLC_PRG.test[269]  +  20  ) * 10.275 + SEL( PLC_PRG.test[269] > 20 , 0.5, -0.5)
  rectangle at (583,214)-(584,224): alarm colour if PLC_PRG.test[270] < 0; top (-1.0 *  PLC_PRG.test[270]  +  20  ) * 10.275 + SEL( PLC_PRG.test[270] > 20 , 0.5, -0.5); bottom (-1.0 *  PLC_PRG.test[270]  +  20  ) * 10.275 + SEL( PLC_PRG.test[270] > 20 , 0.5, -0.5)
  rectangle at (585,214)-(586,224): alarm colour if PLC_PRG.test[271] < 0; top (-1.0 *  PLC_PRG.test[271]  +  20  ) * 10.275 + SEL( PLC_PRG.test[271] > 20 , 0.5, -0.5); bottom (-1.0 *  PLC_PRG.test[271]  +  20  ) * 10.275 + SEL( PLC_PRG.test[271] > 20 , 0.5, -0.5)
  rectangle at (587,214)-(588,224): alarm colour if PLC_PRG.test[272] < 0; top (-1.0 *  PLC_PRG.test[272]  +  20  ) * 10.275 + SEL( PLC_PRG.test[272] > 20 , 0.5, -0.5); bottom (-1.0 *  PLC_PRG.test[272]  +  20  ) * 10.275 + SEL( PLC_PRG.test[272] > 20 , 0.5, -0.5)
  rectangle at (589,214)-(590,224): alarm colour if PLC_PRG.test[273] < 0; top (-1.0 *  PLC_PRG.test[273]  +  20  ) * 10.275 + SEL( PLC_PRG.test[273] > 20 , 0.5, -0.5); bottom (-1.0 *  PLC_PRG.test[273]  +  20  ) * 10.275 + SEL( PLC_PRG.test[273] > 20 , 0.5, -0.5)
  rectangle at (591,214)-(592,224): alarm colour if PLC_PRG.test[274] < 0; top (-1.0 *  PLC_PRG.test[274]  +  20  ) * 10.275 + SEL( PLC_PRG.test[274] > 20 , 0.5, -0.5); bottom (-1.0 *  PLC_PRG.test[274]  +  20  ) * 10.275 + SEL( PLC_PRG.test[274] > 20 , 0.5, -0.5)
  rectangle at (593,214)-(594,224): alarm colour if PLC_PRG.test[275] < 0; top (-1.0 *  PLC_PRG.test[275]  +  20  ) * 10.275 + SEL( PLC_PRG.test[275] > 20 , 0.5, -0.5); bottom (-1.0 *  PLC_PRG.test[275]  +  20  ) * 10.275 + SEL( PLC_PRG.test[275] > 20 , 0.5, -0.5)
  rectangle at (595,214)-(596,224): alarm colour if PLC_PRG.test[276] < 0; top (-1.0 *  PLC_PRG.test[276]  +  20  ) * 10.275 + SEL( PLC_PRG.test[276] > 20 , 0.5, -0.5); bottom (-1.0 *  PLC_PRG.test[276]  +  20  ) * 10.275 + SEL( PLC_PRG.test[276] > 20 , 0.5, -0.5)
  rectangle at (597,214)-(598,224): alarm colour if PLC_PRG.test[277] < 0; top (-1.0 *  PLC_PRG.test[277]  +  20  ) * 10.275 + SEL( PLC_PRG.test[277] > 20 , 0.5, -0.5); bottom (-1.0 *  PLC_PRG.test[277]  +  20  ) * 10.275 + SEL( PLC_PRG.test[277] > 20 , 0.5, -0.5)
  rectangle at (599,214)-(600,224): alarm colour if PLC_PRG.test[278] < 0; top (-1.0 *  PLC_PRG.test[278]  +  20  ) * 10.275 + SEL( PLC_PRG.test[278] > 20 , 0.5, -0.5); bottom (-1.0 *  PLC_PRG.test[278]  +  20  ) * 10.275 + SEL( PLC_PRG.test[278] > 20 , 0.5, -0.5)
  rectangle at (601,214)-(602,224): alarm colour if PLC_PRG.test[279] < 0; top (-1.0 *  PLC_PRG.test[279]  +  20  ) * 10.275 + SEL( PLC_PRG.test[279] > 20 , 0.5, -0.5); bottom (-1.0 *  PLC_PRG.test[279]  +  20  ) * 10.275 + SEL( PLC_PRG.test[279] > 20 , 0.5, -0.5)
  rectangle at (603,214)-(604,224): alarm colour if PLC_PRG.test[280] < 0; top (-1.0 *  PLC_PRG.test[280]  +  20  ) * 10.275 + SEL( PLC_PRG.test[280] > 20 , 0.5, -0.5); bottom (-1.0 *  PLC_PRG.test[280]  +  20  ) * 10.275 + SEL( PLC_PRG.test[280] > 20 , 0.5, -0.5)
  rectangle at (605,214)-(606,224): alarm colour if PLC_PRG.test[281] < 0; top (-1.0 *  PLC_PRG.test[281]  +  20  ) * 10.275 + SEL( PLC_PRG.test[281] > 20 , 0.5, -0.5); bottom (-1.0 *  PLC_PRG.test[281]  +  20  ) * 10.275 + SEL( PLC_PRG.test[281] > 20 , 0.5, -0.5)
  rectangle at (607,214)-(608,224): alarm colour if PLC_PRG.test[282] < 0; top (-1.0 *  PLC_PRG.test[282]  +  20  ) * 10.275 + SEL( PLC_PRG.test[282] > 20 , 0.5, -0.5); bottom (-1.0 *  PLC_PRG.test[282]  +  20  ) * 10.275 + SEL( PLC_PRG.test[282] > 20 , 0.5, -0.5)
  rectangle at (609,214)-(610,224): alarm colour if PLC_PRG.test[283] < 0; top (-1.0 *  PLC_PRG.test[283]  +  20  ) * 10.275 + SEL( PLC_PRG.test[283] > 20 , 0.5, -0.5); bottom (-1.0 *  PLC_PRG.test[283]  +  20  ) * 10.275 + SEL( PLC_PRG.test[283] > 20 , 0.5, -0.5)
  rectangle at (611,214)-(612,224): alarm colour if PLC_PRG.test[284] < 0; top (-1.0 *  PLC_PRG.test[284]  +  20  ) * 10.275 + SEL( PLC_PRG.test[284] > 20 , 0.5, -0.5); bottom (-1.0 *  PLC_PRG.test[284]  +  20  ) * 10.275 + SEL( PLC_PRG.test[284] > 20 , 0.5, -0.5)
  rectangle at (613,214)-(613,224): alarm colour if PLC_PRG.test[285] < 0; top (-1.0 *  PLC_PRG.test[285]  +  20  ) * 10.275 + SEL( PLC_PRG.test[285] > 20 , 0.5, -0.5); bottom (-1.0 *  PLC_PRG.test[285]  +  20  ) * 10.275 + SEL( PLC_PRG.test[285] > 20 , 0.5, -0.5)
  rectangle at (613,214)-(614,224): alarm colour if PLC_PRG.test[286] < 0; top (-1.0 *  PLC_PRG.test[286]  +  20  ) * 10.275 + SEL( PLC_PRG.test[286] > 20 , 0.5, -0.5); bottom (-1.0 *  PLC_PRG.test[286]  +  20  ) * 10.275 + SEL( PLC_PRG.test[286] > 20 , 0.5, -0.5)
  rectangle at (615,214)-(615,224): alarm colour if PLC_PRG.test[287] < 0; top (-1.0 *  PLC_PRG.test[287]  +  20  ) * 10.275 + SEL( PLC_PRG.test[287] > 20 , 0.5, -0.5); bottom (-1.0 *  PLC_PRG.test[287]  +  20  ) * 10.275 + SEL( PLC_PRG.test[287] > 20 , 0.5, -0.5)
  rectangle at (615,214)-(616,224): alarm colour if PLC_PRG.test[288] < 0; top (-1.0 *  PLC_PRG.test[288]  +  20  ) * 10.275 + SEL( PLC_PRG.test[288] > 20 , 0.5, -0.5); bottom (-1.0 *  PLC_PRG.test[288]  +  20  ) * 10.275 + SEL( PLC_PRG.test[288] > 20 , 0.5, -0.5)
  rectangle at (617,214)-(617,224): alarm colour if PLC_PRG.test[289] < 0; top (-1.0 *  PLC_PRG.test[289]  +  20  ) * 10.275 + SEL( PLC_PRG.test[289] > 20 , 0.5, -0.5); bottom (-1.0 *  PLC_PRG.test[289]  +  20  ) * 10.275 + SEL( PLC_PRG.test[289] > 20 , 0.5, -0.5)
  rectangle at (617,214)-(618,224): alarm colour if PLC_PRG.test[290] < 0; top (-1.0 *  PLC_PRG.test[290]  +  20  ) * 10.275 + SEL( PLC_PRG.test[290] > 20 , 0.5, -0.5); bottom (-1.0 *  PLC_PRG.test[290]  +  20  ) * 10.275 + SEL( PLC_PRG.test[290] > 20 , 0.5, -0.5)
  rectangle at (619,214)-(619,224): alarm colour if PLC_PRG.test[291] < 0; top (-1.0 *  PLC_PRG.test[291]  +  20  ) * 10.275 + SEL( PLC_PRG.test[291] > 20 , 0.5, -0.5); bottom (-1.0 *  PLC_PRG.test[291]  +  20  ) * 10.275 + SEL( PLC_PRG.test[291] > 20 , 0.5, -0.5)
  rectangle at (619,214)-(620,224): alarm colour if PLC_PRG.test[292] < 0; top (-1.0 *  PLC_PRG.test[292]  +  20  ) * 10.275 + SEL( PLC_PRG.test[292] > 20 , 0.5, -0.5); bottom (-1.0 *  PLC_PRG.test[292]  +  20  ) * 10.275 + SEL( PLC_PRG.test[292] > 20 , 0.5, -0.5)
  rectangle at (621,214)-(621,224): alarm colour if PLC_PRG.test[293] < 0; top (-1.0 *  PLC_PRG.test[293]  +  20  ) * 10.275 + SEL( PLC_PRG.test[293] > 20 , 0.5, -0.5); bottom (-1.0 *  PLC_PRG.test[293]  +  20  ) * 10.275 + SEL( PLC_PRG.test[293] > 20 , 0.5, -0.5)
  rectangle at (621,214)-(622,224): alarm colour if PLC_PRG.test[294] < 0; top (-1.0 *  PLC_PRG.test[294]  +  20  ) * 10.275 + SEL( PLC_PRG.test[294] > 20 , 0.5, -0.5); bottom (-1.0 *  PLC_PRG.test[294]  +  20  ) * 10.275 + SEL( PLC_PRG.test[294] > 20 , 0.5, -0.5)
  rectangle at (623,214)-(623,224): alarm colour if PLC_PRG.test[295] < 0; top (-1.0 *  PLC_PRG.test[295]  +  20  ) * 10.275 + SEL( PLC_PRG.test[295] > 20 , 0.5, -0.5); bottom (-1.0 *  PLC_PRG.test[295]  +  20  ) * 10.275 + SEL( PLC_PRG.test[295] > 20 , 0.5, -0.5)
  rectangle at (623,214)-(624,224): alarm colour if PLC_PRG.test[296] < 0; top (-1.0 *  PLC_PRG.test[296]  +  20  ) * 10.275 + SEL( PLC_PRG.test[296] > 20 , 0.5, -0.5); bottom (-1.0 *  PLC_PRG.test[296]  +  20  ) * 10.275 + SEL( PLC_PRG.test[296] > 20 , 0.5, -0.5)
  rectangle at (625,214)-(625,224): alarm colour if PLC_PRG.test[297] < 0; top (-1.0 *  PLC_PRG.test[297]  +  20  ) * 10.275 + SEL( PLC_PRG.test[297] > 20 , 0.5, -0.5); bottom (-1.0 *  PLC_PRG.test[297]  +  20  ) * 10.275 + SEL( PLC_PRG.test[297] > 20 , 0.5, -0.5)
  rectangle at (625,214)-(626,224): alarm colour if PLC_PRG.test[298] < 0; top (-1.0 *  PLC_PRG.test[298]  +  20  ) * 10.275 + SEL( PLC_PRG.test[298] > 20 , 0.5, -0.5); bottom (-1.0 *  PLC_PRG.test[298]  +  20  ) * 10.275 + SEL( PLC_PRG.test[298] > 20 , 0.5, -0.5)
  rectangle at (627,214)-(627,224): alarm colour if PLC_PRG.test[299] < 0; top (-1.0 *  PLC_PRG.test[299]  +  20  ) * 10.275 + SEL( PLC_PRG.test[299] > 20 , 0.5, -0.5); bottom (-1.0 *  PLC_PRG.test[299]  +  20  ) * 10.275 + SEL( PLC_PRG.test[299] > 20 , 0.5, -0.5)
  rectangle at (627,214)-(628,224): alarm colour if PLC_PRG.test[300] < 0; top (-1.0 *  PLC_PRG.test[300]  +  20  ) * 10.275 + SEL( PLC_PRG.test[300] > 20 , 0.5, -0.5); bottom (-1.0 *  PLC_PRG.test[300]  +  20  ) * 10.275 + SEL( PLC_PRG.test[300] > 20 , 0.5, -0.5)
  rectangle at (629,214)-(629,224): alarm colour if PLC_PRG.test[301] < 0; top (-1.0 *  PLC_PRG.test[301]  +  20  ) * 10.275 + SEL( PLC_PRG.test[301] > 20 , 0.5, -0.5); bottom (-1.0 *  PLC_PRG.test[301]  +  20  ) * 10.275 + SEL( PLC_PRG.test[301] > 20 , 0.5, -0.5)
  rectangle at (629,214)-(630,224): alarm colour if PLC_PRG.test[302] < 0; top (-1.0 *  PLC_PRG.test[302]  +  20  ) * 10.275 + SEL( PLC_PRG.test[302] > 20 , 0.5, -0.5); bottom (-1.0 *  PLC_PRG.test[302]  +  20  ) * 10.275 + SEL( PLC_PRG.test[302] > 20 , 0.5, -0.5)
  rectangle at (631,214)-(631,224): alarm colour if PLC_PRG.test[303] < 0; top (-1.0 *  PLC_PRG.test[303]  +  20  ) * 10.275 + SEL( PLC_PRG.test[303] > 20 , 0.5, -0.5); bottom (-1.0 *  PLC_PRG.test[303]  +  20  ) * 10.275 + SEL( PLC_PRG.test[303] > 20 , 0.5, -0.5)
  rectangle at (631,214)-(632,224): alarm colour if PLC_PRG.test[304] < 0; top (-1.0 *  PLC_PRG.test[304]  +  20  ) * 10.275 + SEL( PLC_PRG.test[304] > 20 , 0.5, -0.5); bottom (-1.0 *  PLC_PRG.test[304]  +  20  ) * 10.275 + SEL( PLC_PRG.test[304] > 20 , 0.5, -0.5)
  rectangle at (633,214)-(633,224): alarm colour if PLC_PRG.test[305] < 0; top (-1.0 *  PLC_PRG.test[305]  +  20  ) * 10.275 + SEL( PLC_PRG.test[305] > 20 , 0.5, -0.5); bottom (-1.0 *  PLC_PRG.test[305]  +  20  ) * 10.275 + SEL( PLC_PRG.test[305] > 20 , 0.5, -0.5)
  rectangle at (633,214)-(634,224): alarm colour if PLC_PRG.test[306] < 0; top (-1.0 *  PLC_PRG.test[306]  +  20  ) * 10.275 + SEL( PLC_PRG.test[306] > 20 , 0.5, -0.5); bottom (-1.0 *  PLC_PRG.test[306]  +  20  ) * 10.275 + SEL( PLC_PRG.test[306] > 20 , 0.5, -0.5)
  rectangle at (635,214)-(635,224): alarm colour if PLC_PRG.test[307] < 0; top (-1.0 *  PLC_PRG.test[307]  +  20  ) * 10.275 + SEL( PLC_PRG.test[307] > 20 , 0.5, -0.5); bottom (-1.0 *  PLC_PRG.test[307]  +  20  ) * 10.275 + SEL( PLC_PRG.test[307] > 20 , 0.5, -0.5)
  rectangle at (635,214)-(636,224): alarm colour if PLC_PRG.test[308] < 0; top (-1.0 *  PLC_PRG.test[308]  +  20  ) * 10.275 + SEL( PLC_PRG.test[308] > 20 , 0.5, -0.5); bottom (-1.0 *  PLC_PRG.test[308]  +  20  ) * 10.275 + SEL( PLC_PRG.test[308] > 20 , 0.5, -0.5)
  rectangle at (637,214)-(637,224): alarm colour if PLC_PRG.test[309] < 0; top (-1.0 *  PLC_PRG.test[309]  +  20  ) * 10.275 + SEL( PLC_PRG.test[309] > 20 , 0.5, -0.5); bottom (-1.0 *  PLC_PRG.test[309]  +  20  ) * 10.275 + SEL( PLC_PRG.test[309] > 20 , 0.5, -0.5)
  rectangle at (637,214)-(638,224): alarm colour if PLC_PRG.test[310] < 0; top (-1.0 *  PLC_PRG.test[310]  +  20  ) * 10.275 + SEL( PLC_PRG.test[310] > 20 , 0.5, -0.5); bottom (-1.0 *  PLC_PRG.test[310]  +  20  ) * 10.275 + SEL( PLC_PRG.test[310] > 20 , 0.5, -0.5)
  rectangle at (639,214)-(639,224): alarm colour if PLC_PRG.test[311] < 0; top (-1.0 *  PLC_PRG.test[311]  +  20  ) * 10.275 + SEL( PLC_PRG.test[311] > 20 , 0.5, -0.5); bottom (-1.0 *  PLC_PRG.test[311]  +  20  ) * 10.275 + SEL( PLC_PRG.test[311] > 20 , 0.5, -0.5)
  rectangle at (639,214)-(640,224): alarm colour if PLC_PRG.test[312] < 0; top (-1.0 *  PLC_PRG.test[312]  +  20  ) * 10.275 + SEL( PLC_PRG.test[312] > 20 , 0.5, -0.5); bottom (-1.0 *  PLC_PRG.test[312]  +  20  ) * 10.275 + SEL( PLC_PRG.test[312] > 20 , 0.5, -0.5)
  rectangle at (641,214)-(641,224): alarm colour if PLC_PRG.test[313] < 0; top (-1.0 *  PLC_PRG.test[313]  +  20  ) * 10.275 + SEL( PLC_PRG.test[313] > 20 , 0.5, -0.5); bottom (-1.0 *  PLC_PRG.test[313]  +  20  ) * 10.275 + SEL( PLC_PRG.test[313] > 20 , 0.5, -0.5)
  rectangle at (641,214)-(642,224): alarm colour if PLC_PRG.test[314] < 0; top (-1.0 *  PLC_PRG.test[314]  +  20  ) * 10.275 + SEL( PLC_PRG.test[314] > 20 , 0.5, -0.5); bottom (-1.0 *  PLC_PRG.test[314]  +  20  ) * 10.275 + SEL( PLC_PRG.test[314] > 20 , 0.5, -0.5)
  rectangle at (643,214)-(643,224): alarm colour if PLC_PRG.test[315] < 0; top (-1.0 *  PLC_PRG.test[315]  +  20  ) * 10.275 + SEL( PLC_PRG.test[315] > 20 , 0.5, -0.5); bottom (-1.0 *  PLC_PRG.test[315]  +  20  ) * 10.275 + SEL( PLC_PRG.test[315] > 20 , 0.5, -0.5)
  rectangle at (643,214)-(644,224): alarm colour if PLC_PRG.test[316] < 0; top (-1.0 *  PLC_PRG.test[316]  +  20  ) * 10.275 + SEL( PLC_PRG.test[316] > 20 , 0.5, -0.5); bottom (-1.0 *  PLC_PRG.test[316]  +  20  ) * 10.275 + SEL( PLC_PRG.test[316] > 20 , 0.5, -0.5)
  rectangle at (645,214)-(645,224): alarm colour if PLC_PRG.test[317] < 0; top (-1.0 *  PLC_PRG.test[317]  +  20  ) * 10.275 + SEL( PLC_PRG.test[317] > 20 , 0.5, -0.5); bottom (-1.0 *  PLC_PRG.test[317]  +  20  ) * 10.275 + SEL( PLC_PRG.test[317] > 20 , 0.5, -0.5)
  rectangle at (645,214)-(646,224): alarm colour if PLC_PRG.test[318] < 0; top (-1.0 *  PLC_PRG.test[318]  +  20  ) * 10.275 + SEL( PLC_PRG.test[318] > 20 , 0.5, -0.5); bottom (-1.0 *  PLC_PRG.test[318]  +  20  ) * 10.275 + SEL( PLC_PRG.test[318] > 20 , 0.5, -0.5)
  rectangle at (647,214)-(647,224): alarm colour if PLC_PRG.test[319] < 0; top (-1.0 *  PLC_PRG.test[319]  +  20  ) * 10.275 + SEL( PLC_PRG.test[319] > 20 , 0.5, -0.5); bottom (-1.0 *  PLC_PRG.test[319]  +  20  ) * 10.275 + SEL( PLC_PRG.test[319] > 20 , 0.5, -0.5)
  rectangle at (647,214)-(648,224): alarm colour if PLC_PRG.test[320] < 0; top (-1.0 *  PLC_PRG.test[320]  +  20  ) * 10.275 + SEL( PLC_PRG.test[320] > 20 , 0.5, -0.5); bottom (-1.0 *  PLC_PRG.test[320]  +  20  ) * 10.275 + SEL( PLC_PRG.test[320] > 20 , 0.5, -0.5)
  rectangle at (649,214)-(649,224): alarm colour if PLC_PRG.test[321] < 0; top (-1.0 *  PLC_PRG.test[321]  +  20  ) * 10.275 + SEL( PLC_PRG.test[321] > 20 , 0.5, -0.5); bottom (-1.0 *  PLC_PRG.test[321]  +  20  ) * 10.275 + SEL( PLC_PRG.test[321] > 20 , 0.5, -0.5)
  rectangle at (649,214)-(650,224): alarm colour if PLC_PRG.test[322] < 0; top (-1.0 *  PLC_PRG.test[322]  +  20  ) * 10.275 + SEL( PLC_PRG.test[322] > 20 , 0.5, -0.5); bottom (-1.0 *  PLC_PRG.test[322]  +  20  ) * 10.275 + SEL( PLC_PRG.test[322] > 20 , 0.5, -0.5)
  rectangle at (651,214)-(651,224): alarm colour if PLC_PRG.test[323] < 0; top (-1.0 *  PLC_PRG.test[323]  +  20  ) * 10.275 + SEL( PLC_PRG.test[323] > 20 , 0.5, -0.5); bottom (-1.0 *  PLC_PRG.test[323]  +  20  ) * 10.275 + SEL( PLC_PRG.test[323] > 20 , 0.5, -0.5)
  rectangle at (651,214)-(652,224): alarm colour if PLC_PRG.test[324] < 0; top (-1.0 *  PLC_PRG.test[324]  +  20  ) * 10.275 + SEL( PLC_PRG.test[324] > 20 , 0.5, -0.5); bottom (-1.0 *  PLC_PRG.test[324]  +  20  ) * 10.275 + SEL( PLC_PRG.test[324] > 20 , 0.5, -0.5)
  rectangle at (653,214)-(653,224): alarm colour if PLC_PRG.test[325] < 0; top (-1.0 *  PLC_PRG.test[325]  +  20  ) * 10.275 + SEL( PLC_PRG.test[325] > 20 , 0.5, -0.5); bottom (-1.0 *  PLC_PRG.test[325]  +  20  ) * 10.275 + SEL( PLC_PRG.test[325] > 20 , 0.5, -0.5)
  rectangle at (653,214)-(654,224): alarm colour if PLC_PRG.test[326] < 0; top (-1.0 *  PLC_PRG.test[326]  +  20  ) * 10.275 + SEL( PLC_PRG.test[326] > 20 , 0.5, -0.5); bottom (-1.0 *  PLC_PRG.test[326]  +  20  ) * 10.275 + SEL( PLC_PRG.test[326] > 20 , 0.5, -0.5)
  rectangle at (655,214)-(655,224): alarm colour if PLC_PRG.test[327] < 0; top (-1.0 *  PLC_PRG.test[327]  +  20  ) * 10.275 + SEL( PLC_PRG.test[327] > 20 , 0.5, -0.5); bottom (-1.0 *  PLC_PRG.test[327]  +  20  ) * 10.275 + SEL( PLC_PRG.test[327] > 20 , 0.5, -0.5)
  rectangle at (655,214)-(656,224): alarm colour if PLC_PRG.test[328] < 0; top (-1.0 *  PLC_PRG.test[328]  +  20  ) * 10.275 + SEL( PLC_PRG.test[328] > 20 , 0.5, -0.5); bottom (-1.0 *  PLC_PRG.test[328]  +  20  ) * 10.275 + SEL( PLC_PRG.test[328] > 20 , 0.5, -0.5)
  rectangle at (657,214)-(657,224): alarm colour if PLC_PRG.test[329] < 0; top (-1.0 *  PLC_PRG.test[329]  +  20  ) * 10.275 + SEL( PLC_PRG.test[329] > 20 , 0.5, -0.5); bottom (-1.0 *  PLC_PRG.test[329]  +  20  ) * 10.275 + SEL( PLC_PRG.test[329] > 20 , 0.5, -0.5)
  rectangle at (657,214)-(658,224): alarm colour if PLC_PRG.test[330] < 0; top (-1.0 *  PLC_PRG.test[330]  +  20  ) * 10.275 + SEL( PLC_PRG.test[330] > 20 , 0.5, -0.5); bottom (-1.0 *  PLC_PRG.test[330]  +  20  ) * 10.275 + SEL( PLC_PRG.test[330] > 20 , 0.5, -0.5)
  rectangle at (659,214)-(659,224): alarm colour if PLC_PRG.test[331] < 0; top (-1.0 *  PLC_PRG.test[331]  +  20  ) * 10.275 + SEL( PLC_PRG.test[331] > 20 , 0.5, -0.5); bottom (-1.0 *  PLC_PRG.test[331]  +  20  ) * 10.275 + SEL( PLC_PRG.test[331] > 20 , 0.5, -0.5)
  rectangle at (659,214)-(660,224): alarm colour if PLC_PRG.test[332] < 0; top (-1.0 *  PLC_PRG.test[332]  +  20  ) * 10.275 + SEL( PLC_PRG.test[332] > 20 , 0.5, -0.5); bottom (-1.0 *  PLC_PRG.test[332]  +  20  ) * 10.275 + SEL( PLC_PRG.test[332] > 20 , 0.5, -0.5)
  rectangle at (661,214)-(661,224): alarm colour if PLC_PRG.test[333] < 0; top (-1.0 *  PLC_PRG.test[333]  +  20  ) * 10.275 + SEL( PLC_PRG.test[333] > 20 , 0.5, -0.5); bottom (-1.0 *  PLC_PRG.test[333]  +  20  ) * 10.275 + SEL( PLC_PRG.test[333] > 20 , 0.5, -0.5)
  rectangle at (661,214)-(662,224): alarm colour if PLC_PRG.test[334] < 0; top (-1.0 *  PLC_PRG.test[334]  +  20  ) * 10.275 + SEL( PLC_PRG.test[334] > 20 , 0.5, -0.5); bottom (-1.0 *  PLC_PRG.test[334]  +  20  ) * 10.275 + SEL( PLC_PRG.test[334] > 20 , 0.5, -0.5)
  rectangle at (663,214)-(663,224): alarm colour if PLC_PRG.test[335] < 0; top (-1.0 *  PLC_PRG.test[335]  +  20  ) * 10.275 + SEL( PLC_PRG.test[335] > 20 , 0.5, -0.5); bottom (-1.0 *  PLC_PRG.test[335]  +  20  ) * 10.275 + SEL( PLC_PRG.test[335] > 20 , 0.5, -0.5)
  rectangle at (663,214)-(664,224): alarm colour if PLC_PRG.test[336] < 0; top (-1.0 *  PLC_PRG.test[336]  +  20  ) * 10.275 + SEL( PLC_PRG.test[336] > 20 , 0.5, -0.5); bottom (-1.0 *  PLC_PRG.test[336]  +  20  ) * 10.275 + SEL( PLC_PRG.test[336] > 20 , 0.5, -0.5)
  rectangle at (665,214)-(665,224): alarm colour if PLC_PRG.test[337] < 0; top (-1.0 *  PLC_PRG.test[337]  +  20  ) * 10.275 + SEL( PLC_PRG.test[337] > 20 , 0.5, -0.5); bottom (-1.0 *  PLC_PRG.test[337]  +  20  ) * 10.275 + SEL( PLC_PRG.test[337] > 20 , 0.5, -0.5)
  rectangle at (665,214)-(666,224): alarm colour if PLC_PRG.test[338] < 0; top (-1.0 *  PLC_PRG.test[338]  +  20  ) * 10.275 + SEL( PLC_PRG.test[338] > 20 , 0.5, -0.5); bottom (-1.0 *  PLC_PRG.test[338]  +  20  ) * 10.275 + SEL( PLC_PRG.test[338] > 20 , 0.5, -0.5)
  rectangle at (667,214)-(667,224): alarm colour if PLC_PRG.test[339] < 0; top (-1.0 *  PLC_PRG.test[339]  +  20  ) * 10.275 + SEL( PLC_PRG.test[339] > 20 , 0.5, -0.5); bottom (-1.0 *  PLC_PRG.test[339]  +  20  ) * 10.275 + SEL( PLC_PRG.test[339] > 20 , 0.5, -0.5)
  rectangle at (667,214)-(668,224): alarm colour if PLC_PRG.test[340] < 0; top (-1.0 *  PLC_PRG.test[340]  +  20  ) * 10.275 + SEL( PLC_PRG.test[340] > 20 , 0.5, -0.5); bottom (-1.0 *  PLC_PRG.test[340]  +  20  ) * 10.275 + SEL( PLC_PRG.test[340] > 20 , 0.5, -0.5)
  rectangle at (669,214)-(669,224): alarm colour if PLC_PRG.test[341] < 0; top (-1.0 *  PLC_PRG.test[341]  +  20  ) * 10.275 + SEL( PLC_PRG.test[341] > 20 , 0.5, -0.5); bottom (-1.0 *  PLC_PRG.test[341]  +  20  ) * 10.275 + SEL( PLC_PRG.test[341] > 20 , 0.5, -0.5)
  rectangle at (669,214)-(670,224): alarm colour if PLC_PRG.test[342] < 0; top (-1.0 *  PLC_PRG.test[342]  +  20  ) * 10.275 + SEL( PLC_PRG.test[342] > 20 , 0.5, -0.5); bottom (-1.0 *  PLC_PRG.test[342]  +  20  ) * 10.275 + SEL( PLC_PRG.test[342] > 20 , 0.5, -0.5)
  rectangle at (671,214)-(671,224): alarm colour if PLC_PRG.test[343] < 0; top (-1.0 *  PLC_PRG.test[343]  +  20  ) * 10.275 + SEL( PLC_PRG.test[343] > 20 , 0.5, -0.5); bottom (-1.0 *  PLC_PRG.test[343]  +  20  ) * 10.275 + SEL( PLC_PRG.test[343] > 20 , 0.5, -0.5)
  rectangle at (671,214)-(672,224): alarm colour if PLC_PRG.test[344] < 0; top (-1.0 *  PLC_PRG.test[344]  +  20  ) * 10.275 + SEL( PLC_PRG.test[344] > 20 , 0.5, -0.5); bottom (-1.0 *  PLC_PRG.test[344]  +  20  ) * 10.275 + SEL( PLC_PRG.test[344] > 20 , 0.5, -0.5)
  rectangle at (673,214)-(673,224): alarm colour if PLC_PRG.test[345] < 0; top (-1.0 *  PLC_PRG.test[345]  +  20  ) * 10.275 + SEL( PLC_PRG.test[345] > 20 , 0.5, -0.5); bottom (-1.0 *  PLC_PRG.test[345]  +  20  ) * 10.275 + SEL( PLC_PRG.test[345] > 20 , 0.5, -0.5)
  rectangle at (673,214)-(674,224): alarm colour if PLC_PRG.test[346] < 0; top (-1.0 *  PLC_PRG.test[346]  +  20  ) * 10.275 + SEL( PLC_PRG.test[346] > 20 , 0.5, -0.5); bottom (-1.0 *  PLC_PRG.test[346]  +  20  ) * 10.275 + SEL( PLC_PRG.test[346] > 20 , 0.5, -0.5)
  rectangle at (675,214)-(675,224): alarm colour if PLC_PRG.test[347] < 0; top (-1.0 *  PLC_PRG.test[347]  +  20  ) * 10.275 + SEL( PLC_PRG.test[347] > 20 , 0.5, -0.5); bottom (-1.0 *  PLC_PRG.test[347]  +  20  ) * 10.275 + SEL( PLC_PRG.test[347] > 20 , 0.5, -0.5)
  rectangle at (675,214)-(676,224): alarm colour if PLC_PRG.test[348] < 0; top (-1.0 *  PLC_PRG.test[348]  +  20  ) * 10.275 + SEL( PLC_PRG.test[348] > 20 , 0.5, -0.5); bottom (-1.0 *  PLC_PRG.test[348]  +  20  ) * 10.275 + SEL( PLC_PRG.test[348] > 20 , 0.5, -0.5)
  rectangle at (677,214)-(677,224): alarm colour if PLC_PRG.test[349] < 0; top (-1.0 *  PLC_PRG.test[349]  +  20  ) * 10.275 + SEL( PLC_PRG.test[349] > 20 , 0.5, -0.5); bottom (-1.0 *  PLC_PRG.test[349]  +  20  ) * 10.275 + SEL( PLC_PRG.test[349] > 20 , 0.5, -0.5)
  rectangle at (677,214)-(678,224): alarm colour if PLC_PRG.test[350] < 0; top (-1.0 *  PLC_PRG.test[350]  +  20  ) * 10.275 + SEL( PLC_PRG.test[350] > 20 , 0.5, -0.5); bottom (-1.0 *  PLC_PRG.test[350]  +  20  ) * 10.275 + SEL( PLC_PRG.test[350] > 20 , 0.5, -0.5)
  rectangle at (679,214)-(679,224): alarm colour if PLC_PRG.test[351] < 0; top (-1.0 *  PLC_PRG.test[351]  +  20  ) * 10.275 + SEL( PLC_PRG.test[351] > 20 , 0.5, -0.5); bottom (-1.0 *  PLC_PRG.test[351]  +  20  ) * 10.275 + SEL( PLC_PRG.test[351] > 20 , 0.5, -0.5)
  rectangle at (679,214)-(680,224): alarm colour if PLC_PRG.test[352] < 0; top (-1.0 *  PLC_PRG.test[352]  +  20  ) * 10.275 + SEL( PLC_PRG.test[352] > 20 , 0.5, -0.5); bottom (-1.0 *  PLC_PRG.test[352]  +  20  ) * 10.275 + SEL( PLC_PRG.test[352] > 20 , 0.5, -0.5)
  rectangle at (681,214)-(681,224): alarm colour if PLC_PRG.test[353] < 0; top (-1.0 *  PLC_PRG.test[353]  +  20  ) * 10.275 + SEL( PLC_PRG.test[353] > 20 , 0.5, -0.5); bottom (-1.0 *  PLC_PRG.test[353]  +  20  ) * 10.275 + SEL( PLC_PRG.test[353] > 20 , 0.5, -0.5)
  rectangle at (681,214)-(682,224): alarm colour if PLC_PRG.test[354] < 0; top (-1.0 *  PLC_PRG.test[354]  +  20  ) * 10.275 + SEL( PLC_PRG.test[354] > 20 , 0.5, -0.5); bottom (-1.0 *  PLC_PRG.test[354]  +  20  ) * 10.275 + SEL( PLC_PRG.test[354] > 20 , 0.5, -0.5)
  rectangle at (683,214)-(683,224): alarm colour if PLC_PRG.test[355] < 0; top (-1.0 *  PLC_PRG.test[355]  +  20  ) * 10.275 + SEL( PLC_PRG.test[355] > 20 , 0.5, -0.5); bottom (-1.0 *  PLC_PRG.test[355]  +  20  ) * 10.275 + SEL( PLC_PRG.test[355] > 20 , 0.5, -0.5)
  rectangle at (683,214)-(684,224): alarm colour if PLC_PRG.test[356] < 0; top (-1.0 *  PLC_PRG.test[356]  +  20  ) * 10.275 + SEL( PLC_PRG.test[356] > 20 , 0.5, -0.5); bottom (-1.0 *  PLC_PRG.test[356]  +  20  ) * 10.275 + SEL( PLC_PRG.test[356] > 20 , 0.5, -0.5)
  rectangle at (685,214)-(685,224): alarm colour if PLC_PRG.test[357] < 0; top (-1.0 *  PLC_PRG.test[357]  +  20  ) * 10.275 + SEL( PLC_PRG.test[357] > 20 , 0.5, -0.5); bottom (-1.0 *  PLC_PRG.test[357]  +  20  ) * 10.275 + SEL( PLC_PRG.test[357] > 20 , 0.5, -0.5)
  rectangle at (685,214)-(686,224): alarm colour if PLC_PRG.test[358] < 0; top (-1.0 *  PLC_PRG.test[358]  +  20  ) * 10.275 + SEL( PLC_PRG.test[358] > 20 , 0.5, -0.5); bottom (-1.0 *  PLC_PRG.test[358]  +  20  ) * 10.275 + SEL( PLC_PRG.test[358] > 20 , 0.5, -0.5)
  rectangle at (687,214)-(687,224): alarm colour if PLC_PRG.test[359] < 0; top (-1.0 *  PLC_PRG.test[359]  +  20  ) * 10.275 + SEL( PLC_PRG.test[359] > 20 , 0.5, -0.5); bottom (-1.0 *  PLC_PRG.test[359]  +  20  ) * 10.275 + SEL( PLC_PRG.test[359] > 20 , 0.5, -0.5)
  rectangle at (687,214)-(688,224): alarm colour if PLC_PRG.test[360] < 0; top (-1.0 *  PLC_PRG.test[360]  +  20  ) * 10.275 + SEL( PLC_PRG.test[360] > 20 , 0.5, -0.5); bottom (-1.0 *  PLC_PRG.test[360]  +  20  ) * 10.275 + SEL( PLC_PRG.test[360] > 20 , 0.5, -0.5)
85 more shapes without text or variables
*)
